C05431=1052.907,134.284,-84.781,171.313,33.859,156.345
C05432=1052.901,134.035,-84.760,171.311,33.857,156.345
C05433=1052.896,133.786,-84.739,171.310,33.854,156.344
C05434=1052.889,133.537,-84.718,171.307,33.852,156.344
C05435=1052.884,133.288,-84.697,171.305,33.850,156.344
C05436=1052.878,133.038,-84.676,171.303,33.847,156.343
C05437=1052.871,132.790,-84.656,171.301,33.845,156.343
C05438=1052.866,132.540,-84.635,171.300,33.843,156.342
C05439=1052.860,132.292,-84.613,171.298,33.841,156.342
C05440=1052.853,132.042,-84.593,171.296,33.838,156.342
C05441=1052.848,131.794,-84.572,171.294,33.836,156.341
C05442=1052.842,131.544,-84.551,171.293,33.834,156.341
C05443=1052.836,131.296,-84.530,171.291,33.832,156.340
C05444=1052.829,131.046,-84.510,171.289,33.829,156.340
C05445=1052.824,130.797,-84.489,171.287,33.827,156.340
C05446=1052.817,130.548,-84.468,171.286,33.825,156.339
C05447=1052.812,130.299,-84.448,171.284,33.823,156.339
C05448=1052.805,130.049,-84.427,171.282,33.821,156.339
C05449=1052.799,129.801,-84.407,171.280,33.818,156.338
C05450=1052.793,129.551,-84.386,171.279,33.816,156.338
C05451=1052.786,129.303,-84.365,171.277,33.814,156.337
C05452=1052.780,129.054,-84.345,171.275,33.812,156.337
C05453=1052.774,128.804,-84.324,171.273,33.809,156.337
C05454=1052.768,128.556,-84.303,171.271,33.807,156.336
C05455=1052.761,128.306,-84.283,171.269,33.806,156.336
C05456=1052.756,128.057,-84.262,171.267,33.803,156.336
C05457=1052.750,127.808,-84.242,171.265,33.801,156.335
C05458=1052.744,127.559,-84.221,171.263,33.798,156.335
C05459=1052.738,127.310,-84.201,171.262,33.797,156.334
C05460=1052.731,127.061,-84.180,171.260,33.794,156.334
C05461=1052.726,126.812,-84.159,171.258,33.792,156.334
C05462=1052.719,126.563,-84.139,171.257,33.790,156.333
C05463=1052.712,126.277,-84.115,171.255,33.788,156.333
C05464=1052.705,125.991,-84.092,171.253,33.785,156.332
C05465=1052.698,125.706,-84.069,171.251,33.782,156.332
C05466=1052.692,125.421,-84.045,171.249,33.780,156.332
C05467=1052.685,125.172,-84.025,171.247,33.777,156.331
C05468=1052.679,124.924,-84.004,171.245,33.775,156.331
C05469=1052.673,124.674,-83.983,171.243,33.773,156.330
C05470=1052.667,124.425,-83.963,171.242,33.771,156.330
C05471=1052.661,124.175,-83.943,171.240,33.768,156.330
C05472=1052.655,123.926,-83.923,171.238,33.766,156.329
C05473=1052.649,123.677,-83.903,171.236,33.764,156.329
C05474=1052.643,123.429,-83.882,171.235,33.762,156.328
C05475=1052.637,123.179,-83.861,171.232,33.760,156.328
C05476=1052.631,122.930,-83.841,171.230,33.757,156.328
C05477=1052.625,122.681,-83.821,171.229,33.755,156.327
C05478=1052.619,122.432,-83.801,171.227,33.753,156.327
C05479=1052.613,122.182,-83.780,171.225,33.751,156.327
C05480=1052.607,121.934,-83.760,171.223,33.748,156.326
C05481=1052.601,121.685,-83.740,171.222,33.746,156.326
C05482=1052.595,121.436,-83.718,171.220,33.744,156.325
C05483=1052.589,121.187,-83.698,171.218,33.742,156.325
C05484=1052.583,120.938,-83.678,171.217,33.739,156.325
C05485=1052.577,120.688,-83.657,171.215,33.737,156.324
C05486=1052.571,120.439,-83.637,171.213,33.735,156.324
C05487=1052.565,120.191,-83.617,171.211,33.733,156.324
C05488=1052.558,119.941,-83.597,171.210,33.731,156.323
C05489=1052.553,119.692,-83.577,171.208,33.728,156.323
C05490=1052.547,119.443,-83.557,171.206,33.726,156.322
C05491=1052.540,119.194,-83.536,171.205,33.724,156.322
C05492=1052.535,118.944,-83.516,171.203,33.722,156.322
C05493=1052.529,118.696,-83.496,171.201,33.719,156.321
C05494=1052.523,118.447,-83.476,171.200,33.718,156.321
C05495=1052.517,118.197,-83.456,171.198,33.715,156.321
C05496=1052.511,117.948,-83.435,171.196,33.713,156.320
C05497=1052.505,117.699,-83.415,171.194,33.710,156.320
C05498=1052.499,117.450,-83.395,171.192,33.708,156.319
C05499=1052.493,117.201,-83.374,171.190,33.706,156.319
C05500=1052.487,116.952,-83.354,171.188,33.704,156.319
C05501=1052.481,116.703,-83.334,171.187,33.701,156.318
C05502=1052.475,116.454,-83.314,171.185,33.699,156.318
C05503=1052.470,116.204,-83.294,171.183,33.697,156.317
C05504=1052.464,115.955,-83.274,171.182,33.695,156.317
C05505=1052.458,115.706,-83.254,171.180,33.692,156.317
C05506=1052.451,115.457,-83.234,171.178,33.690,156.316
C05507=1052.446,115.208,-83.213,171.177,33.688,156.316
C05508=1052.440,114.959,-83.193,171.175,33.686,156.316
C05509=1052.434,114.710,-83.173,171.173,33.683,156.315
C05510=1052.428,114.461,-83.153,171.172,33.682,156.315
C05511=1052.423,114.211,-83.133,171.170,33.679,156.314
C05512=1052.417,113.962,-83.113,171.168,33.677,156.314
C05513=1052.411,113.713,-83.093,171.167,33.674,156.314
C05514=1052.405,113.464,-83.073,171.165,33.672,156.313
C05515=1052.398,113.215,-83.053,171.163,33.670,156.313
C05516=1052.392,112.965,-83.034,171.161,33.668,156.313
C05517=1052.386,112.717,-83.014,171.160,33.666,156.312
C05518=1052.380,112.468,-82.994,171.158,33.663,156.312
C05519=1052.374,112.218,-82.973,171.156,33.661,156.311
C05520=1052.368,111.969,-82.954,171.155,33.659,156.311
C05521=1052.362,111.720,-82.934,171.153,33.657,156.311
C05522=1052.356,111.471,-82.914,171.151,33.655,156.310
C05523=1052.350,111.222,-82.894,171.149,33.653,156.310
C05524=1052.344,110.972,-82.875,171.147,33.651,156.310
C05525=1052.338,110.723,-82.855,171.145,33.648,156.309
C05526=1052.332,110.475,-82.835,171.144,33.646,156.309
C05527=1052.324,110.189,-82.813,171.142,33.643,156.308
C05528=1052.318,109.903,-82.790,171.140,33.641,156.308
C05529=1052.311,109.618,-82.768,171.138,33.639,156.308
C05530=1052.303,109.332,-82.745,171.136,33.636,156.307
C05531=1052.297,109.083,-82.725,171.134,33.634,156.307
C05532=1052.292,108.834,-82.706,171.133,33.632,156.306
C05533=1052.285,108.584,-82.686,171.131,33.630,156.306
C05534=1052.279,108.336,-82.666,171.129,33.627,156.306
C05535=1052.273,108.086,-82.647,171.128,33.625,156.305
C05536=1052.267,107.838,-82.627,171.126,33.623,156.305
C05537=1052.261,107.588,-82.608,171.124,33.621,156.305
C05538=1052.254,107.339,-82.588,171.123,33.619,156.304
C05539=1052.248,107.090,-82.568,171.121,33.617,156.304
C05540=1052.243,106.840,-82.548,171.119,33.614,156.304
C05541=1052.237,106.592,-82.528,171.117,33.612,156.303
C05542=1052.230,106.343,-82.510,171.116,33.610,156.303
C05543=1052.224,106.094,-82.490,171.114,33.608,156.302
C05544=1052.218,105.844,-82.470,171.112,33.606,156.302
C05545=1052.212,105.595,-82.450,171.111,33.603,156.302
C05546=1052.206,105.345,-82.431,171.109,33.601,156.301
C05547=1052.200,105.096,-82.411,171.108,33.600,156.301
C05548=1052.194,104.847,-82.392,171.106,33.597,156.301
C05549=1052.188,104.599,-82.372,171.104,33.595,156.300
C05550=1052.182,104.349,-82.353,171.103,33.593,156.300
C05551=1052.176,104.100,-82.333,171.101,33.590,156.299
C05552=1052.170,103.850,-82.314,171.098,33.589,156.299
C05553=1052.163,103.602,-82.294,171.097,33.586,156.299
C05554=1052.158,103.352,-82.275,171.095,33.584,156.298
C05555=1052.152,103.103,-82.255,171.093,33.582,156.298
C05556=1052.146,102.854,-82.236,171.092,33.580,156.298
C05557=1052.140,102.605,-82.217,171.090,33.578,156.297
C05558=1052.133,102.356,-82.197,171.088,33.576,156.297
C05559=1052.128,102.107,-82.178,171.087,33.573,156.297
C05560=1052.122,101.858,-82.158,171.085,33.571,156.296
C05561=1052.116,101.608,-82.139,171.083,33.568,156.296
C05562=1052.110,101.359,-82.120,171.082,33.567,156.295
C05563=1052.104,101.110,-82.100,171.080,33.565,156.295
C05564=1052.098,100.861,-82.081,171.078,33.562,156.295
C05565=1052.092,100.611,-82.061,171.077,33.560,156.294
C05566=1052.086,100.362,-82.041,171.075,33.558,156.294
C05567=1052.079,100.113,-82.023,171.073,33.556,156.294
C05568=1052.074,99.864,-82.003,171.072,33.554,156.293
C05569=1052.067,99.615,-81.984,171.070,33.552,156.293
C05570=1052.061,99.366,-81.965,171.068,33.549,156.293
C05571=1052.055,99.116,-81.946,171.067,33.547,156.292
C05572=1052.049,98.867,-81.927,171.065,33.545,156.292
C05573=1052.042,98.619,-81.908,171.063,33.543,156.292
C05574=1052.037,98.369,-81.888,171.062,33.541,156.291
C05575=1052.031,98.120,-81.869,171.060,33.539,156.291
C05576=1052.024,97.871,-81.850,171.059,33.537,156.291
C05577=1052.018,97.621,-81.830,171.057,33.534,156.290
C05578=1052.011,97.372,-81.811,171.055,33.532,156.290
C05579=1052.006,97.122,-81.792,171.054,33.530,156.289
C05580=1051.999,96.873,-81.774,171.052,33.528,156.289
C05581=1051.994,96.624,-81.754,171.050,33.526,156.289
C05582=1051.987,96.375,-81.735,171.049,33.524,156.288
C05583=1051.981,96.126,-81.716,171.047,33.522,156.288
C05584=1051.975,95.877,-81.697,171.045,33.519,156.288
C05585=1051.969,95.627,-81.678,171.044,33.517,156.287
C05586=1051.963,95.378,-81.659,171.042,33.515,156.287
C05587=1051.957,95.129,-81.639,171.040,33.513,156.287
C05588=1051.951,94.880,-81.620,171.038,33.511,156.286
C05589=1051.945,94.631,-81.601,171.036,33.509,156.286
C05590=1051.939,94.382,-81.582,171.034,33.506,156.285
C05591=1051.932,94.096,-81.561,171.033,33.504,156.285
C05592=1051.925,93.810,-81.538,171.031,33.502,156.285
C05593=1051.918,93.525,-81.517,171.029,33.499,156.284
C05594=1051.912,93.240,-81.495,171.027,33.497,156.284
C05595=1051.905,92.990,-81.477,171.025,33.495,156.283
C05596=1051.899,92.741,-81.457,171.024,33.493,156.283
C05597=1051.893,92.492,-81.439,171.022,33.490,156.283
C05598=1051.887,92.242,-81.419,171.020,33.488,156.282
C05599=1051.881,91.994,-81.400,171.019,33.486,156.282
C05600=1051.875,91.745,-81.381,171.017,33.484,156.282
C05601=1051.868,91.495,-81.362,171.016,33.482,156.281
C05602=1051.863,91.246,-81.343,171.014,33.480,156.281
C05603=1051.856,90.997,-81.324,171.012,33.477,156.281
C05604=1051.851,90.747,-81.305,171.011,33.475,156.280
C05605=1051.844,90.498,-81.286,171.009,33.473,156.280
C05606=1051.838,90.249,-81.268,171.007,33.471,156.280
C05607=1051.832,90.000,-81.249,171.006,33.469,156.279
C05608=1051.826,89.750,-81.231,171.004,33.467,156.279
C05609=1051.820,89.501,-81.212,171.002,33.465,156.279
C05610=1051.813,89.252,-81.193,171.001,33.463,156.278
C05611=1051.807,89.002,-81.174,170.999,33.460,156.278
C05612=1051.802,88.754,-81.156,170.998,33.458,156.277
C05613=1051.795,88.505,-81.137,170.996,33.456,156.277
C05614=1051.789,88.256,-81.118,170.994,33.454,156.277
C05615=1051.783,88.006,-81.099,170.993,33.452,156.276
C05616=1051.777,87.757,-81.081,170.991,33.450,156.276
C05617=1051.770,87.508,-81.062,170.989,33.448,156.276
C05618=1051.764,87.259,-81.043,170.988,33.446,156.275
C05619=1051.758,87.009,-81.025,170.986,33.444,156.275
C05620=1051.752,86.760,-81.006,170.984,33.441,156.275
C05621=1051.746,86.511,-80.987,170.983,33.439,156.274
C05622=1051.739,86.261,-80.969,170.981,33.437,156.274
C05623=1051.733,86.012,-80.950,170.979,33.435,156.274
C05624=1051.727,85.763,-80.931,170.978,33.433,156.273
C05625=1051.722,85.514,-80.913,170.976,33.431,156.273
C05626=1051.715,85.265,-80.895,170.975,33.429,156.273
C05627=1051.709,85.016,-80.876,170.973,33.427,156.272
C05628=1051.703,84.766,-80.857,170.971,33.424,156.272
C05629=1051.697,84.517,-80.838,170.970,33.422,156.272
C05630=1051.690,84.267,-80.820,170.968,33.420,156.271
C05631=1051.684,84.018,-80.802,170.966,33.418,156.271
C05632=1051.678,83.769,-80.782,170.965,33.416,156.270
C05633=1051.672,83.520,-80.764,170.963,33.414,156.270
C05634=1051.666,83.271,-80.746,170.962,33.412,156.270
C05635=1051.660,83.021,-80.727,170.960,33.410,156.270
C05636=1051.654,82.772,-80.709,170.958,33.407,156.269
C05637=1051.648,82.523,-80.690,170.957,33.405,156.269
C05638=1051.642,82.273,-80.672,170.954,33.403,156.268
C05639=1051.636,82.025,-80.653,170.952,33.401,156.268
C05640=1051.629,81.776,-80.635,170.951,33.399,156.268
C05641=1051.623,81.526,-80.617,170.949,33.397,156.267
C05642=1051.618,81.276,-80.598,170.948,33.395,156.267
C05643=1051.611,81.027,-80.579,170.946,33.392,156.267
C05644=1051.606,80.778,-80.561,170.944,33.390,156.266
C05645=1051.599,80.529,-80.543,170.943,33.389,156.266
C05646=1051.593,80.280,-80.524,170.941,33.387,156.266
C05647=1051.587,80.030,-80.506,170.939,33.384,156.265
C05648=1051.581,79.781,-80.487,170.938,33.382,156.265
C05649=1051.575,79.532,-80.469,170.936,33.380,156.265
C05650=1051.569,79.283,-80.451,170.935,33.378,156.264
C05651=1051.563,79.034,-80.432,170.933,33.375,156.264
C05652=1051.557,78.784,-80.414,170.931,33.373,156.264
C05653=1051.551,78.535,-80.396,170.930,33.372,156.263
C05654=1051.545,78.286,-80.377,170.928,33.369,156.263
C05655=1051.538,78.001,-80.356,170.926,33.367,156.262
C05656=1051.530,77.715,-80.335,170.924,33.364,156.262
C05657=1051.524,77.428,-80.314,170.923,33.362,156.262
C05658=1051.516,77.143,-80.294,170.921,33.360,156.261
C05659=1051.510,76.894,-80.275,170.919,33.358,156.261
C05660=1051.504,76.645,-80.257,170.917,33.355,156.261
C05661=1051.498,76.396,-80.239,170.916,33.353,156.260
C05662=1051.492,76.146,-80.221,170.914,33.351,156.260
C05663=1051.485,75.897,-80.202,170.913,33.349,156.260
C05664=1051.479,75.647,-80.184,170.911,33.347,156.259
C05665=1051.474,75.399,-80.166,170.909,33.345,156.259
C05666=1051.467,75.149,-80.148,170.908,33.343,156.259
C05667=1051.461,74.900,-80.129,170.906,33.341,156.258
C05668=1051.455,74.650,-80.111,170.904,33.339,156.258
C05669=1051.449,74.402,-80.093,170.903,33.337,156.258
C05670=1051.443,74.152,-80.075,170.901,33.335,156.257
C05671=1051.436,73.903,-80.058,170.900,33.332,156.257
C05672=1051.430,73.654,-80.039,170.898,33.330,156.257
C05673=1051.424,73.404,-80.022,170.896,33.328,156.256
C05674=1051.418,73.155,-80.003,170.895,33.326,156.256
C05675=1051.412,72.906,-79.985,170.893,33.324,156.256
C05676=1051.406,72.657,-79.967,170.891,33.322,156.255
C05677=1051.400,72.407,-79.949,170.890,33.320,156.255
C05678=1051.394,72.158,-79.931,170.888,33.318,156.254
C05679=1051.387,71.909,-79.912,170.887,33.316,156.254
C05680=1051.382,71.660,-79.895,170.885,33.314,156.254
C05681=1051.375,71.410,-79.877,170.883,33.311,156.253
C05682=1051.368,71.161,-79.859,170.882,33.309,156.253
C05683=1051.363,70.912,-79.841,170.880,33.307,156.253
C05684=1051.357,70.662,-79.823,170.878,33.305,156.252
C05685=1051.350,70.413,-79.805,170.877,33.304,156.252
C05686=1051.345,70.164,-79.787,170.875,33.301,156.252
C05687=1051.339,69.914,-79.769,170.874,33.299,156.251
C05688=1051.332,69.665,-79.750,170.872,33.297,156.251
C05689=1051.326,69.416,-79.733,170.870,33.295,156.251
C05690=1051.320,69.167,-79.716,170.869,33.293,156.250
C05691=1051.314,68.917,-79.698,170.867,33.291,156.250
C05692=1051.308,68.669,-79.679,170.865,33.288,156.250
C05693=1051.301,68.419,-79.662,170.864,33.287,156.249
C05694=1051.295,68.169,-79.644,170.862,33.285,156.249
C05695=1051.289,67.920,-79.626,170.861,33.283,156.249
C05696=1051.283,67.671,-79.609,170.859,33.281,156.248
C05697=1051.276,67.422,-79.591,170.857,33.279,156.248
C05698=1051.271,67.173,-79.573,170.856,33.277,156.248
C05699=1051.264,66.923,-79.555,170.854,33.274,156.247
C05700=1051.258,66.673,-79.537,170.852,33.272,156.247
C05701=1051.252,66.425,-79.520,170.851,33.270,156.247
C05702=1051.246,66.175,-79.501,170.849,33.268,156.246
C05703=1051.240,65.926,-79.484,170.847,33.266,156.246
C05704=1051.233,65.677,-79.467,170.846,33.264,156.246
C05705=1051.227,65.427,-79.449,170.844,33.262,156.245
C05706=1051.222,65.178,-79.431,170.843,33.260,156.245
C05707=1051.215,64.929,-79.414,170.841,33.258,156.245
C05708=1051.209,64.679,-79.396,170.839,33.256,156.244
C05709=1051.203,64.430,-79.378,170.838,33.254,156.244
C05710=1051.197,64.181,-79.360,170.836,33.252,156.244
C05711=1051.190,63.932,-79.343,170.834,33.250,156.243
C05712=1051.184,63.683,-79.325,170.833,33.248,156.243
C05713=1051.177,63.433,-79.307,170.831,33.246,156.243
C05714=1051.171,63.184,-79.290,170.830,33.244,156.243
C05715=1051.165,62.934,-79.272,170.828,33.242,156.242
C05716=1051.158,62.685,-79.255,170.826,33.240,156.242
C05717=1051.153,62.436,-79.238,170.825,33.238,156.242
C05718=1051.146,62.187,-79.220,170.823,33.236,156.241
C05719=1051.139,61.901,-79.200,170.821,33.233,156.241
C05720=1051.132,61.615,-79.180,170.819,33.231,156.241
C05721=1051.124,61.330,-79.160,170.817,33.229,156.240
C05722=1051.117,61.044,-79.140,170.815,33.227,156.240
C05723=1051.111,60.794,-79.122,170.814,33.225,156.239
C05724=1051.105,60.545,-79.105,170.812,33.223,156.239
C05725=1051.098,60.296,-79.087,170.810,33.221,156.239
C05726=1051.092,60.046,-79.070,170.809,33.219,156.239
C05727=1051.085,59.797,-79.053,170.807,33.217,156.238
C05728=1051.080,59.547,-79.036,170.806,33.215,156.238
C05729=1051.073,59.298,-79.019,170.804,33.213,156.238
C05730=1051.067,59.049,-79.001,170.802,33.211,156.237
C05731=1051.061,58.800,-78.984,170.801,33.208,156.237
C05732=1051.054,58.550,-78.967,170.799,33.206,156.237
C05733=1051.048,58.301,-78.949,170.797,33.204,156.236
C05734=1051.042,58.052,-78.932,170.796,33.202,156.236
C05735=1051.036,57.802,-78.914,170.794,33.200,156.236
C05736=1051.029,57.553,-78.897,170.792,33.198,156.235
C05737=1051.023,57.303,-78.880,170.791,33.196,156.235
C05738=1051.017,57.054,-78.863,170.789,33.194,156.235
C05739=1051.010,56.805,-78.845,170.787,33.192,156.234
C05740=1051.005,56.556,-78.828,170.786,33.190,156.234
C05741=1050.998,56.306,-78.810,170.784,33.188,156.234
C05742=1050.992,56.058,-78.793,170.783,33.186,156.233
C05743=1050.986,55.807,-78.776,170.781,33.184,156.233
C05744=1050.980,55.559,-78.759,170.779,33.182,156.233
C05745=1050.974,55.309,-78.741,170.778,33.180,156.232
C05746=1050.967,55.060,-78.724,170.776,33.178,156.232
C05747=1050.960,54.811,-78.707,170.774,33.176,156.232
C05748=1050.955,54.561,-78.690,170.773,33.174,156.231
C05749=1050.948,54.312,-78.673,170.771,33.172,156.231
C05750=1050.943,54.063,-78.655,170.769,33.170,156.231
C05751=1050.936,53.813,-78.638,170.768,33.168,156.230
C05752=1050.930,53.564,-78.622,170.766,33.166,156.230
C05753=1050.924,53.314,-78.604,170.765,33.164,156.230
C05754=1050.918,53.065,-78.587,170.763,33.162,156.229
C05755=1050.911,52.816,-78.569,170.761,33.160,156.229
C05756=1050.906,52.566,-78.553,170.760,33.158,156.229
C05757=1050.899,52.317,-78.535,170.758,33.156,156.229
C05758=1050.892,52.068,-78.518,170.756,33.154,156.228
C05759=1050.887,51.818,-78.501,170.755,33.152,156.228
C05760=1050.880,51.569,-78.484,170.753,33.150,156.228
C05761=1050.875,51.320,-78.467,170.751,33.148,156.227
C05762=1050.868,51.070,-78.450,170.750,33.146,156.227
C05763=1050.862,50.821,-78.433,170.748,33.144,156.227
C05764=1050.856,50.571,-78.415,170.747,33.141,156.226
C05765=1050.850,50.322,-78.399,170.745,33.139,156.226
C05766=1050.844,50.073,-78.382,170.743,33.137,156.226
C05767=1050.838,49.824,-78.364,170.742,33.136,156.225
C05768=1050.832,49.574,-78.348,170.740,33.133,156.225
C05769=1050.825,49.325,-78.330,170.738,33.131,156.225
C05770=1050.819,49.076,-78.313,170.737,33.130,156.224
C05771=1050.813,48.827,-78.296,170.735,33.128,156.224
C05772=1050.806,48.577,-78.279,170.733,33.125,156.224
C05773=1050.801,48.327,-78.262,170.732,33.124,156.223
C05774=1050.795,48.079,-78.245,170.730,33.122,156.223
C05775=1050.788,47.829,-78.228,170.728,33.119,156.223
C05776=1050.783,47.580,-78.211,170.727,33.117,156.222
C05777=1050.777,47.331,-78.194,170.725,33.115,156.222
C05778=1050.770,47.081,-78.177,170.724,33.113,156.222
C05779=1050.765,46.832,-78.160,170.722,33.111,156.221
C05780=1050.759,46.582,-78.144,170.720,33.109,156.221
C05781=1050.752,46.333,-78.126,170.719,33.107,156.221
C05782=1050.747,46.083,-78.109,170.717,33.105,156.220
C05783=1050.739,45.798,-78.090,170.715,33.102,156.220
C05784=1050.732,45.511,-78.071,170.713,33.100,156.220
C05785=1050.725,45.225,-78.051,170.711,33.098,156.219
C05786=1050.718,44.939,-78.032,170.710,33.095,156.219
C05787=1050.712,44.690,-78.015,170.708,33.093,156.219
C05788=1050.706,44.441,-77.998,170.706,33.091,156.218
C05789=1050.700,44.191,-77.981,170.705,33.089,156.218
C05790=1050.694,43.942,-77.964,170.703,33.087,156.218
C05791=1050.688,43.693,-77.947,170.701,33.085,156.217
C05792=1050.682,43.443,-77.931,170.700,33.083,156.217
C05793=1050.675,43.194,-77.914,170.698,33.081,156.217
C05794=1050.669,42.945,-77.897,170.696,33.079,156.216
C05795=1050.663,42.695,-77.881,170.695,33.077,156.216
C05796=1050.656,42.446,-77.864,170.693,33.075,156.216
C05797=1050.651,42.197,-77.848,170.691,33.073,156.215
C05798=1050.645,41.947,-77.831,170.690,33.071,156.215
C05799=1050.638,41.697,-77.813,170.688,33.069,156.215
C05800=1050.632,41.448,-77.797,170.686,33.067,156.215
C05801=1050.627,41.199,-77.781,170.685,33.065,156.214
C05802=1050.620,40.949,-77.764,170.683,33.063,156.214
C05803=1050.614,40.700,-77.747,170.681,33.061,156.214
C05804=1050.608,40.451,-77.731,170.680,33.059,156.213
C05805=1050.602,40.202,-77.714,170.678,33.057,156.213
C05806=1050.595,39.952,-77.697,170.676,33.055,156.213
C05807=1050.589,39.702,-77.681,170.675,33.053,156.212
C05808=1050.583,39.454,-77.664,170.673,33.051,156.212
C05809=1050.576,39.204,-77.648,170.671,33.049,156.212
C05810=1050.570,38.954,-77.631,170.670,33.047,156.211
C05811=1050.564,38.705,-77.615,170.668,33.045,156.211
C05812=1050.558,38.456,-77.598,170.667,33.043,156.211
C05813=1050.551,38.206,-77.581,170.665,33.041,156.211
C05814=1050.546,37.957,-77.565,170.663,33.039,156.210
C05815=1050.540,37.708,-77.549,170.662,33.037,156.210
C05816=1050.533,37.459,-77.532,170.660,33.035,156.210
C05817=1050.527,37.209,-77.515,170.658,33.033,156.209
C05818=1050.521,36.959,-77.499,170.657,33.031,156.209
C05819=1050.515,36.710,-77.483,170.655,33.029,156.209
C05820=1050.509,36.461,-77.467,170.653,33.027,156.208
C05821=1050.502,36.211,-77.450,170.651,33.025,156.208
C05822=1050.495,35.962,-77.434,170.650,33.024,156.208
C05823=1050.489,35.713,-77.417,170.648,33.022,156.208
C05824=1050.483,35.464,-77.401,170.646,33.020,156.207
C05825=1050.477,35.213,-77.384,170.645,33.018,156.207
C05826=1050.471,34.964,-77.368,170.644,33.016,156.207
C05827=1050.465,34.715,-77.352,170.642,33.014,156.206
C05828=1050.458,34.466,-77.336,170.641,33.012,156.206
C05829=1050.452,34.216,-77.320,170.639,33.010,156.206
C05830=1050.446,33.967,-77.303,170.637,33.008,156.205
C05831=1050.440,33.718,-77.286,170.636,33.006,156.205
C05832=1050.434,33.468,-77.270,170.634,33.004,156.205
C05833=1050.428,33.219,-77.254,170.632,33.002,156.205
C05834=1050.420,32.969,-77.238,170.631,33.001,156.204
C05835=1050.414,32.720,-77.222,170.629,32.998,156.204
C05836=1050.408,32.471,-77.205,170.627,32.996,156.204
C05837=1050.403,32.221,-77.189,170.626,32.995,156.203
C05838=1050.397,31.972,-77.173,170.624,32.992,156.203
C05839=1050.390,31.723,-77.157,170.622,32.990,156.203
C05840=1050.383,31.473,-77.141,170.621,32.988,156.202
C05841=1050.377,31.223,-77.124,170.619,32.986,156.202
C05842=1050.371,30.974,-77.108,170.617,32.984,156.202
C05843=1050.365,30.725,-77.092,170.615,32.983,156.202
C05844=1050.359,30.476,-77.076,170.614,32.981,156.201
C05845=1050.353,30.226,-77.060,170.612,32.979,156.201
C05846=1050.346,29.976,-77.043,170.610,32.977,156.201
C05847=1050.340,29.691,-77.025,170.609,32.974,156.200
C05848=1050.332,29.404,-77.006,170.607,32.972,156.200
C05849=1050.325,29.119,-76.988,170.605,32.970,156.200
C05850=1050.318,28.833,-76.969,170.603,32.968,156.199
C05851=1050.312,28.583,-76.953,170.601,32.966,156.199
C05852=1050.306,28.333,-76.938,170.599,32.964,156.199
C05853=1050.299,28.084,-76.922,170.598,32.962,156.198
C05854=1050.293,27.834,-76.905,170.596,32.960,156.198
C05855=1050.287,27.585,-76.889,170.594,32.958,156.198
C05856=1050.280,27.336,-76.873,170.593,32.956,156.197
C05857=1050.274,27.087,-76.857,170.591,32.955,156.197
C05858=1050.269,26.837,-76.841,170.589,32.953,156.197
C05859=1050.262,26.588,-76.825,170.587,32.951,156.197
C05860=1050.256,26.338,-76.810,170.586,32.949,156.196
C05861=1050.250,26.088,-76.793,170.584,32.947,156.196
C05862=1050.243,25.839,-76.777,170.582,32.945,156.196
C05863=1050.237,25.590,-76.761,170.581,32.943,156.196
C05864=1050.230,25.341,-76.746,170.579,32.941,156.195
C05865=1050.225,25.091,-76.730,170.577,32.939,156.195
C05866=1050.218,24.842,-76.714,170.576,32.937,156.195
C05867=1050.212,24.592,-76.698,170.574,32.935,156.194
C05868=1050.206,24.343,-76.682,170.572,32.934,156.194
C05869=1050.199,24.094,-76.666,170.570,32.932,156.194
C05870=1050.194,23.844,-76.651,170.569,32.930,156.193
C05871=1050.186,23.594,-76.635,170.567,32.928,156.193
C05872=1050.181,23.345,-76.618,170.565,32.926,156.193
C05873=1050.174,23.096,-76.603,170.564,32.924,156.193
C05874=1050.168,22.846,-76.587,170.562,32.923,156.192
C05875=1050.162,22.597,-76.571,170.560,32.920,156.192
C05876=1050.156,22.348,-76.555,170.558,32.918,156.192
C05877=1050.150,22.098,-76.540,170.558,32.917,156.191
C05878=1050.143,21.849,-76.524,170.556,32.914,156.191
C05879=1050.137,21.599,-76.508,170.554,32.913,156.191
C05880=1050.131,21.350,-76.493,170.553,32.911,156.191
C05881=1050.125,21.100,-76.477,170.551,32.909,156.190
C05882=1050.118,20.851,-76.461,170.549,32.907,156.190
C05883=1050.113,20.601,-76.445,170.547,32.905,156.190
C05884=1050.106,20.352,-76.430,170.546,32.904,156.190
C05885=1050.100,20.103,-76.413,170.544,32.902,156.189
C05886=1050.094,19.853,-76.398,170.542,32.900,156.189
C05887=1050.088,19.604,-76.382,170.541,32.898,156.189
C05888=1050.081,19.355,-76.367,170.539,32.896,156.188
C05889=1050.075,19.105,-76.351,170.537,32.894,156.188
C05890=1050.069,18.856,-76.335,170.535,32.892,156.188
C05891=1050.063,18.606,-76.320,170.534,32.890,156.187
C05892=1050.056,18.357,-76.304,170.532,32.888,156.187
C05893=1050.050,18.107,-76.289,170.530,32.887,156.187
C05894=1050.044,17.858,-76.273,170.528,32.885,156.187
C05895=1050.037,17.609,-76.257,170.527,32.883,156.186
C05896=1050.032,17.359,-76.242,170.525,32.881,156.186
C05897=1050.025,17.110,-76.226,170.523,32.879,156.186
C05898=1050.019,16.860,-76.211,170.522,32.877,156.186
C05899=1050.013,16.611,-76.195,170.520,32.875,156.185
C05900=1050.006,16.361,-76.180,170.518,32.873,156.185
C05901=1050.000,16.112,-76.164,170.516,32.872,156.185
C05902=1049.994,15.862,-76.149,170.515,32.870,156.184
C05903=1049.987,15.613,-76.133,170.513,32.868,156.184
C05904=1049.982,15.363,-76.118,170.511,32.866,156.184
C05905=1049.975,15.114,-76.102,170.509,32.864,156.184
C05906=1049.968,14.864,-76.087,170.508,32.862,156.183
C05907=1049.962,14.615,-76.071,170.506,32.860,156.183
C05908=1049.956,14.365,-76.056,170.504,32.858,156.183
C05909=1049.950,14.115,-76.040,170.502,32.857,156.183
C05910=1049.944,13.866,-76.024,170.501,32.855,156.182
C05911=1049.937,13.582,-76.007,170.499,32.853,156.182
C05912=1049.929,13.297,-75.990,170.497,32.851,156.182
C05913=1049.922,13.012,-75.972,170.495,32.849,156.181
C05914=1049.915,12.728,-75.955,170.493,32.847,156.181
C05915=1049.909,12.478,-75.940,170.491,32.845,156.181
C05916=1049.902,12.229,-75.924,170.490,32.843,156.181
C05917=1049.896,11.979,-75.909,170.488,32.841,156.180
C05918=1049.890,11.730,-75.894,170.487,32.840,156.180
C05919=1049.883,11.481,-75.879,170.485,32.838,156.180
C05920=1049.877,11.231,-75.864,170.483,32.836,156.179
C05921=1049.871,10.981,-75.848,170.481,32.834,156.179
C05922=1049.864,10.732,-75.833,170.480,32.832,156.179
C05923=1049.858,10.482,-75.818,170.478,32.831,156.179
C05924=1049.851,10.233,-75.803,170.476,32.829,156.178
C05925=1049.845,9.983,-75.788,170.474,32.827,156.178
C05926=1049.838,9.734,-75.772,170.472,32.825,156.178
C05927=1049.832,9.484,-75.757,170.471,32.823,156.178
C05928=1049.827,9.235,-75.742,170.469,32.822,156.177
C05929=1049.820,8.986,-75.726,170.467,32.820,156.177
C05930=1049.814,8.736,-75.711,170.465,32.818,156.177
C05931=1049.807,8.487,-75.696,170.464,32.817,156.177
C05932=1049.801,8.237,-75.681,170.462,32.814,156.176
C05933=1049.795,7.987,-75.666,170.460,32.812,156.176
C05934=1049.788,7.738,-75.651,170.458,32.811,156.176
C05935=1049.782,7.489,-75.636,170.457,32.809,156.176
C05936=1049.777,7.239,-75.621,170.455,32.808,156.175
C05937=1049.770,6.990,-75.606,170.453,32.806,156.175
C05938=1049.764,6.740,-75.591,170.451,32.803,156.175
C05939=1049.757,6.491,-75.575,170.449,32.802,156.175
C05940=1049.751,6.241,-75.560,170.448,32.800,156.174
C05941=1049.744,5.992,-75.545,170.446,32.799,156.174
C05942=1049.739,5.743,-75.531,170.444,32.797,156.174
C05943=1049.732,5.493,-75.516,170.442,32.795,156.174
C05944=1049.726,5.243,-75.501,170.441,32.793,156.173
C05945=1049.719,4.994,-75.485,170.439,32.791,156.173
C05946=1049.713,4.744,-75.470,170.437,32.789,156.173
C05947=1049.707,4.495,-75.455,170.435,32.788,156.173
C05948=1049.701,4.246,-75.440,170.434,32.786,156.172
C05949=1049.695,3.996,-75.425,170.433,32.784,156.172
C05950=1049.689,3.746,-75.410,170.431,32.782,156.172
C05951=1049.682,3.497,-75.395,170.429,32.780,156.171
C05952=1049.676,3.248,-75.381,170.427,32.779,156.171
C05953=1049.670,2.998,-75.366,170.426,32.777,156.171
C05954=1049.664,2.749,-75.351,170.424,32.775,156.171
C05955=1049.657,2.499,-75.336,170.422,32.773,156.170
C05956=1049.651,2.250,-75.321,170.420,32.771,156.170
C05957=1049.645,2.001,-75.306,170.418,32.770,156.170
C05958=1049.638,1.751,-75.291,170.417,32.768,156.170
C05959=1049.633,1.501,-75.275,170.415,32.766,156.169
C05960=1049.627,1.252,-75.261,170.413,32.764,156.169
C05961=1049.621,1.003,-75.246,170.411,32.762,156.169
C05962=1049.614,0.753,-75.231,170.409,32.761,156.169
C05963=1049.608,0.503,-75.216,170.408,32.759,156.168
C05964=1049.602,0.254,-75.201,170.406,32.757,156.168
C05965=1049.596,0.005,-75.186,170.404,32.755,156.168
C05966=1049.589,-0.245,-75.171,170.402,32.753,156.168
C05967=1049.584,-0.495,-75.157,170.400,32.752,156.167
C05968=1049.577,-0.744,-75.142,170.399,32.750,156.167
C05969=1049.571,-0.994,-75.127,170.397,32.748,156.167
C05970=1049.565,-1.244,-75.112,170.395,32.746,156.167
C05971=1049.559,-1.492,-75.098,170.393,32.744,156.166
C05972=1049.552,-1.742,-75.083,170.392,32.743,156.166
C05973=1049.546,-1.992,-75.068,170.390,32.741,156.166
C05974=1049.540,-2.241,-75.053,170.388,32.739,156.166
C05975=1049.533,-2.524,-75.036,170.386,32.737,156.165
C05976=1049.527,-2.807,-75.020,170.384,32.735,156.165
C05977=1049.520,-3.090,-75.003,170.383,32.733,156.165
C05978=1049.513,-3.373,-74.986,170.381,32.731,156.164
C05979=1049.507,-3.622,-74.972,170.379,32.729,156.164
C05980=1049.500,-3.871,-74.957,170.377,32.728,156.164
C05981=1049.493,-4.121,-74.942,170.375,32.726,156.164
C05982=1049.487,-4.371,-74.928,170.373,32.724,156.163
C05983=1049.482,-4.620,-74.914,170.372,32.723,156.163
C05984=1049.474,-4.870,-74.899,170.370,32.721,156.163
C05985=1049.468,-5.119,-74.884,170.368,32.719,156.163
C05986=1049.462,-5.368,-74.870,170.366,32.717,156.162
C05987=1049.456,-5.618,-74.855,170.364,32.716,156.162
C05988=1049.449,-5.868,-74.841,170.362,32.714,156.162
C05989=1049.443,-6.117,-74.827,170.361,32.713,156.162
C05990=1049.437,-6.366,-74.812,170.359,32.711,156.162
C05991=1049.430,-6.616,-74.798,170.357,32.709,156.161
C05992=1049.424,-6.865,-74.783,170.355,32.708,156.161
C05993=1049.418,-7.115,-74.769,170.353,32.706,156.161
C05994=1049.412,-7.365,-74.754,170.351,32.704,156.161
C05995=1049.405,-7.614,-74.740,170.350,32.703,156.160
C05996=1049.399,-7.864,-74.725,170.348,32.701,156.160
C05997=1049.393,-8.113,-74.710,170.346,32.699,156.160
C05998=1049.386,-8.362,-74.697,170.344,32.697,156.160
C05999=1049.380,-8.612,-74.682,170.342,32.696,156.160
C06000=1049.374,-8.861,-74.668,170.340,32.694,156.159
C06001=1049.368,-9.111,-74.653,170.338,32.692,156.159
C06002=1049.361,-9.361,-74.639,170.337,32.691,156.159
C06003=1049.355,-9.610,-74.624,170.336,32.689,156.159
C06004=1049.349,-9.860,-74.610,170.334,32.687,156.158
C06005=1049.342,-10.109,-74.596,170.332,32.686,156.158
C06006=1049.336,-10.358,-74.581,170.330,32.684,156.158
C06007=1049.330,-10.608,-74.567,170.328,32.682,156.158
C06008=1049.324,-10.857,-74.553,170.327,32.680,156.157
C06009=1049.318,-11.107,-74.539,170.325,32.679,156.157
C06010=1049.312,-11.356,-74.524,170.323,32.678,156.157
C06011=1049.306,-11.607,-74.510,170.321,32.675,156.157
C06012=1049.299,-11.856,-74.496,170.319,32.674,156.157
C06013=1049.293,-12.105,-74.481,170.317,32.672,156.156
C06014=1049.287,-12.355,-74.467,170.315,32.671,156.156
C06015=1049.280,-12.604,-74.453,170.314,32.669,156.156
C06016=1049.274,-12.854,-74.439,170.312,32.667,156.156
C06017=1049.268,-13.103,-74.424,170.310,32.666,156.155
C06018=1049.262,-13.353,-74.410,170.308,32.664,156.155
C06019=1049.256,-13.602,-74.396,170.306,32.662,156.155
C06020=1049.250,-13.852,-74.382,170.304,32.661,156.155
C06021=1049.243,-14.101,-74.368,170.302,32.659,156.154
C06022=1049.237,-14.351,-74.353,170.301,32.657,156.154
C06023=1049.231,-14.600,-74.339,170.299,32.656,156.154
C06024=1049.224,-14.850,-74.325,170.297,32.654,156.154
C06025=1049.219,-15.099,-74.311,170.295,32.652,156.154
C06026=1049.212,-15.349,-74.297,170.293,32.650,156.153
C06027=1049.206,-15.599,-74.283,170.292,32.649,156.153
C06028=1049.199,-15.848,-74.269,170.290,32.647,156.153
C06029=1049.193,-16.098,-74.255,170.288,32.646,156.153
C06030=1049.187,-16.347,-74.241,170.286,32.644,156.152
C06031=1049.181,-16.597,-74.226,170.285,32.643,156.152
C06032=1049.174,-16.846,-74.213,170.283,32.641,156.152
C06033=1049.168,-17.096,-74.198,170.281,32.640,156.152
C06034=1049.162,-17.345,-74.185,170.279,32.638,156.152
C06035=1049.155,-17.595,-74.171,170.277,32.636,156.151
C06036=1049.149,-17.844,-74.157,170.275,32.635,156.151
C06037=1049.142,-18.094,-74.143,170.273,32.633,156.151
C06038=1049.137,-18.343,-74.128,170.271,32.632,156.151
C06039=1049.130,-18.584,-74.116,170.270,32.630,156.151
C06040=1049.125,-18.825,-74.102,170.268,32.628,156.150
C06041=1049.118,-19.066,-74.089,170.266,32.627,156.150
C06042=1049.112,-19.307,-74.075,170.264,32.625,156.150
C06043=1049.106,-19.548,-74.062,170.262,32.624,156.150
C06044=1049.100,-19.788,-74.048,170.260,32.623,156.150
C06045=1049.094,-20.029,-74.035,170.259,32.621,156.149
C06046=1049.088,-20.270,-74.022,170.257,32.619,156.149
C06047=1049.081,-20.519,-74.008,170.255,32.618,156.149
C06048=1049.075,-20.769,-73.994,170.253,32.616,156.149
C06049=1049.069,-21.019,-73.980,170.251,32.615,156.149
C06050=1049.064,-21.268,-73.966,170.249,32.613,156.148
C06051=1049.056,-21.518,-73.952,170.248,32.611,156.148
C06052=1049.050,-21.767,-73.939,170.246,32.610,156.148
C06053=1049.044,-22.017,-73.925,170.244,32.608,156.148
C06054=1049.038,-22.266,-73.911,170.242,32.607,156.148
C06055=1049.032,-22.516,-73.896,170.241,32.606,156.147
C06056=1049.025,-22.765,-73.883,170.239,32.603,156.147
C06057=1049.019,-23.015,-73.870,170.237,32.602,156.147
C06058=1049.013,-23.265,-73.856,170.235,32.601,156.147
C06059=1049.007,-23.514,-73.842,170.233,32.599,156.147
C06060=1049.001,-23.764,-73.828,170.231,32.598,156.146
C06061=1048.994,-24.013,-73.814,170.229,32.596,156.146
C06062=1048.988,-24.262,-73.801,170.227,32.594,156.146
C06063=1048.982,-24.513,-73.787,170.225,32.593,156.146
C06064=1048.976,-24.762,-73.773,170.223,32.591,156.146
C06065=1048.970,-25.011,-73.760,170.221,32.590,156.145
C06066=1048.963,-25.261,-73.746,170.219,32.588,156.145
C06067=1048.957,-25.511,-73.733,170.218,32.586,156.145
C06068=1048.951,-25.760,-73.719,170.216,32.585,156.145
C06069=1048.945,-26.010,-73.704,170.214,32.583,156.144
C06070=1048.938,-26.259,-73.691,170.212,32.582,156.144
C06071=1048.933,-26.508,-73.677,170.210,32.580,156.144
C06072=1048.926,-26.758,-73.664,170.208,32.578,156.144
C06073=1048.920,-27.008,-73.650,170.207,32.577,156.144
C06074=1048.914,-27.257,-73.637,170.205,32.576,156.143
C06075=1048.907,-27.507,-73.623,170.203,32.574,156.143
C06076=1048.901,-27.756,-73.609,170.201,32.573,156.143
C06077=1048.895,-28.006,-73.596,170.199,32.571,156.143
C06078=1048.888,-28.256,-73.583,170.197,32.570,156.143
C06079=1048.882,-28.505,-73.569,170.195,32.568,156.143
C06080=1048.876,-28.754,-73.556,170.193,32.567,156.142
C06081=1048.869,-29.004,-73.542,170.191,32.565,156.142
C06082=1048.863,-29.253,-73.529,170.189,32.564,156.142
C06083=1048.857,-29.503,-73.515,170.187,32.562,156.142
C06084=1048.851,-29.753,-73.502,170.186,32.561,156.142
C06085=1048.845,-30.003,-73.489,170.184,32.560,156.141
C06086=1048.839,-30.252,-73.476,170.182,32.558,156.141
C06087=1048.832,-30.502,-73.462,170.180,32.557,156.141
C06088=1048.826,-30.751,-73.449,170.178,32.555,156.141
C06089=1048.819,-31.001,-73.436,170.176,32.554,156.141
C06090=1048.812,-31.251,-73.422,170.174,32.552,156.141
C06091=1048.806,-31.500,-73.409,170.172,32.551,156.140
C06092=1048.801,-31.749,-73.395,170.170,32.549,156.140
C06093=1048.795,-31.999,-73.382,170.168,32.548,156.140
C06094=1048.788,-32.249,-73.368,170.167,32.546,156.140
C06095=1048.782,-32.498,-73.355,170.165,32.545,156.140
C06096=1048.776,-32.748,-73.342,170.163,32.544,156.139
C06097=1048.769,-32.997,-73.329,170.161,32.542,156.139
C06098=1048.763,-33.247,-73.315,170.159,32.541,156.139
C06099=1048.756,-33.496,-73.302,170.157,32.539,156.139
C06100=1048.750,-33.745,-73.289,170.155,32.538,156.139
C06101=1048.744,-33.995,-73.276,170.153,32.536,156.139
C06102=1048.736,-34.343,-73.257,170.150,32.534,156.138
C06103=1048.726,-34.723,-73.237,170.147,32.532,156.138
C06104=1048.719,-35.003,-73.222,170.145,32.530,156.138
C06105=1048.712,-35.283,-73.207,170.143,32.528,156.138
C06106=1048.705,-35.564,-73.192,170.141,32.527,156.137
C06107=1048.698,-35.813,-73.179,170.139,32.525,156.137
C06108=1048.693,-36.063,-73.166,170.137,32.524,156.137
C06109=1048.686,-36.312,-73.153,170.135,32.522,156.137
C06110=1048.680,-36.562,-73.140,170.133,32.521,156.137
C06111=1048.674,-36.812,-73.127,170.131,32.520,156.137
C06112=1048.667,-37.062,-73.114,170.129,32.518,156.136
C06113=1048.662,-37.311,-73.100,170.127,32.517,156.136
C06114=1048.656,-37.560,-73.086,170.126,32.515,156.136
C06115=1048.650,-37.810,-73.074,170.124,32.514,156.136
C06116=1048.644,-38.060,-73.061,170.122,32.513,156.136
C06117=1048.637,-38.309,-73.047,170.120,32.511,156.136
C06118=1048.631,-38.559,-73.034,170.118,32.510,156.135
C06119=1048.625,-38.809,-73.021,170.116,32.508,156.135
C06120=1048.619,-39.059,-73.009,170.114,32.507,156.135
C06121=1048.612,-39.307,-72.996,170.112,32.506,156.135
C06122=1048.606,-39.557,-72.983,170.110,32.504,156.135
C06123=1048.600,-39.807,-72.970,170.108,32.503,156.135
C06124=1048.593,-40.057,-72.956,170.106,32.502,156.134
C06125=1048.587,-40.306,-72.944,170.104,32.500,156.134
C06126=1048.581,-40.556,-72.931,170.102,32.499,156.134
C06127=1048.574,-40.805,-72.918,170.100,32.497,156.134
C06128=1048.568,-41.055,-72.905,170.098,32.496,156.134
C06129=1048.562,-41.304,-72.892,170.096,32.495,156.134
C06130=1048.556,-41.554,-72.880,170.094,32.494,156.133
C06131=1048.549,-41.804,-72.866,170.092,32.492,156.133
C06132=1048.542,-42.053,-72.854,170.090,32.491,156.133
C06133=1048.536,-42.302,-72.841,170.088,32.490,156.133
C06134=1048.530,-42.552,-72.828,170.087,32.488,156.133
C06135=1048.524,-42.802,-72.815,170.085,32.487,156.133
C06136=1048.518,-43.052,-72.802,170.083,32.485,156.133
C06137=1048.511,-43.300,-72.790,170.081,32.484,156.132
C06138=1048.505,-43.550,-72.777,170.079,32.483,156.132
C06139=1048.499,-43.800,-72.764,170.077,32.482,156.132
C06140=1048.492,-44.050,-72.751,170.075,32.480,156.132
C06141=1048.486,-44.299,-72.738,170.073,32.479,156.132
C06142=1048.480,-44.549,-72.726,170.071,32.478,156.132
C06143=1048.474,-44.799,-72.713,170.069,32.476,156.131
C06144=1048.467,-45.048,-72.700,170.066,32.475,156.131
C06145=1048.462,-45.298,-72.687,170.064,32.473,156.131
C06146=1048.455,-45.547,-72.674,170.062,32.473,156.131
C06147=1048.449,-45.797,-72.662,170.060,32.471,156.131
C06148=1048.443,-46.047,-72.650,170.058,32.470,156.131
C06149=1048.437,-46.296,-72.636,170.056,32.468,156.131
C06150=1048.431,-46.546,-72.624,170.054,32.467,156.130
C06151=1048.424,-46.795,-72.611,170.052,32.466,156.130
C06152=1048.418,-47.045,-72.598,170.050,32.464,156.130
C06153=1048.412,-47.295,-72.586,170.049,32.463,156.130
C06154=1048.406,-47.544,-72.573,170.047,32.462,156.130
C06155=1048.400,-47.794,-72.560,170.045,32.461,156.130
C06156=1048.393,-48.043,-72.548,170.043,32.459,156.130
C06157=1048.387,-48.293,-72.535,170.041,32.458,156.129
C06158=1048.381,-48.543,-72.522,170.039,32.457,156.129
C06159=1048.375,-48.792,-72.510,170.037,32.455,156.129
C06160=1048.368,-49.041,-72.497,170.035,32.454,156.129
C06161=1048.362,-49.291,-72.485,170.033,32.453,156.129
C06162=1048.356,-49.541,-72.472,170.031,32.452,156.129
C06163=1048.350,-49.791,-72.459,170.029,32.450,156.129
C06164=1048.343,-50.040,-72.447,170.027,32.449,156.128
C06165=1048.338,-50.290,-72.434,170.025,32.448,156.128
C06166=1048.332,-50.540,-72.422,170.023,32.446,156.128
C06167=1048.324,-50.820,-72.408,170.020,32.445,156.128
C06168=1048.317,-51.102,-72.394,170.018,32.444,156.128
C06169=1048.310,-51.382,-72.380,170.016,32.442,156.128
C06170=1048.303,-51.663,-72.366,170.013,32.441,156.128
C06171=1048.297,-51.913,-72.354,170.011,32.440,156.127
C06172=1048.290,-52.162,-72.342,170.010,32.439,156.127
C06173=1048.284,-52.412,-72.329,170.008,32.438,156.127
C06174=1048.277,-52.662,-72.317,170.006,32.437,156.127
C06175=1048.271,-52.911,-72.305,170.004,32.435,156.127
C06176=1048.265,-53.161,-72.293,170.002,32.435,156.127
C06177=1048.258,-53.411,-72.281,170.000,32.433,156.127
C06178=1048.252,-53.660,-72.267,169.998,32.432,156.127
C06179=1048.245,-53.909,-72.256,169.995,32.431,156.127
C06180=1048.239,-54.159,-72.244,169.993,32.430,156.126
C06181=1048.233,-54.409,-72.231,169.991,32.428,156.126
C06182=1048.226,-54.658,-72.219,169.989,32.428,156.126
C06183=1048.220,-54.908,-72.206,169.987,32.426,156.126
C06184=1048.214,-55.158,-72.195,169.985,32.425,156.126
C06185=1048.207,-55.407,-72.183,169.983,32.424,156.126
C06186=1048.201,-55.657,-72.170,169.981,32.423,156.126
C06187=1048.194,-55.907,-72.158,169.979,32.422,156.126
C06188=1048.189,-56.157,-72.145,169.977,32.421,156.126
C06189=1048.182,-56.406,-72.134,169.975,32.420,156.125
C06190=1048.175,-56.656,-72.122,169.972,32.418,156.125
C06191=1048.169,-56.906,-72.109,169.971,32.417,156.125
C06192=1048.163,-57.155,-72.097,169.969,32.416,156.125
C06193=1048.157,-57.404,-72.085,169.967,32.415,156.125
C06194=1048.151,-57.654,-72.073,169.965,32.414,156.125
C06195=1048.144,-57.904,-72.061,169.963,32.413,156.125
C06196=1048.138,-58.154,-72.048,169.961,32.412,156.125
C06197=1048.132,-58.403,-72.036,169.959,32.411,156.125
C06198=1048.125,-58.653,-72.024,169.957,32.409,156.124
C06199=1048.119,-58.903,-72.012,169.955,32.409,156.124
C06200=1048.113,-59.152,-72.000,169.952,32.407,156.124
C06201=1048.106,-59.401,-71.988,169.950,32.406,156.124
C06202=1048.100,-59.651,-71.976,169.948,32.405,156.124
C06203=1048.094,-59.901,-71.964,169.946,32.404,156.124
C06204=1048.087,-60.151,-71.953,169.944,32.403,156.124
C06205=1048.081,-60.401,-71.940,169.942,32.402,156.124
C06206=1048.075,-60.650,-71.928,169.940,32.401,156.124
C06207=1048.069,-60.899,-71.917,169.938,32.400,156.124
C06208=1048.063,-61.149,-71.904,169.936,32.398,156.123
C06209=1048.056,-61.399,-71.892,169.933,32.397,156.123
C06210=1048.050,-61.648,-71.880,169.932,32.397,156.123
C06211=1048.045,-61.898,-71.869,169.930,32.395,156.123
C06212=1048.038,-62.147,-71.857,169.928,32.394,156.123
C06213=1048.031,-62.397,-71.845,169.926,32.393,156.123
C06214=1048.025,-62.647,-71.832,169.924,32.392,156.123
C06215=1048.019,-62.897,-71.820,169.922,32.391,156.123
C06216=1048.013,-63.145,-71.809,169.920,32.390,156.123
C06217=1048.007,-63.396,-71.797,169.917,32.389,156.123
C06218=1048.000,-63.645,-71.785,169.915,32.388,156.122
C06219=1047.994,-63.895,-71.773,169.913,32.386,156.122
C06220=1047.988,-64.144,-71.761,169.911,32.385,156.122
C06221=1047.982,-64.394,-71.749,169.909,32.385,156.122
C06222=1047.976,-64.644,-71.737,169.907,32.383,156.122
C06223=1047.970,-64.894,-71.725,169.905,32.382,156.122
C06224=1047.964,-65.143,-71.713,169.903,32.381,156.122
C06225=1047.957,-65.393,-71.702,169.901,32.380,156.122
C06226=1047.951,-65.642,-71.690,169.898,32.379,156.122
C06227=1047.945,-65.892,-71.678,169.896,32.378,156.122
C06228=1047.939,-66.142,-71.667,169.894,32.377,156.122
C06229=1047.932,-66.391,-71.655,169.893,32.376,156.121
C06230=1047.926,-66.641,-71.642,169.891,32.375,156.121
C06231=1047.920,-66.923,-71.629,169.888,32.374,156.121
C06232=1047.912,-67.205,-71.616,169.886,32.373,156.121
C06233=1047.906,-67.488,-71.603,169.884,32.372,156.121
C06234=1047.899,-67.770,-71.590,169.881,32.370,156.121
C06235=1047.893,-68.020,-71.577,169.879,32.369,156.121
C06236=1047.886,-68.270,-71.566,169.877,32.368,156.121
C06237=1047.880,-68.519,-71.554,169.875,32.367,156.121
C06238=1047.874,-68.769,-71.543,169.873,32.366,156.121
C06239=1047.868,-69.019,-71.530,169.871,32.365,156.120
C06240=1047.862,-69.268,-71.519,169.868,32.364,156.120
C06241=1047.856,-69.518,-71.508,169.866,32.363,156.120
C06242=1047.850,-69.767,-71.496,169.864,32.362,156.120
C06243=1047.844,-70.017,-71.484,169.862,32.361,156.120
C06244=1047.837,-70.267,-71.472,169.860,32.360,156.120
C06245=1047.831,-70.516,-71.461,169.858,32.359,156.120
C06246=1047.825,-70.766,-71.449,169.856,32.358,156.120
C06247=1047.819,-71.016,-71.437,169.854,32.357,156.120
C06248=1047.813,-71.265,-71.426,169.852,32.356,156.120
C06249=1047.807,-71.515,-71.414,169.850,32.355,156.120
C06250=1047.801,-71.764,-71.403,169.848,32.354,156.119
C06251=1047.795,-72.014,-71.391,169.846,32.353,156.119
C06252=1047.789,-72.264,-71.380,169.844,32.352,156.119
C06253=1047.783,-72.513,-71.368,169.842,32.351,156.119
C06254=1047.776,-72.763,-71.356,169.839,32.350,156.119
C06255=1047.771,-73.013,-71.344,169.837,32.349,156.119
C06256=1047.765,-73.263,-71.333,169.835,32.348,156.119
C06257=1047.759,-73.512,-71.321,169.833,32.347,156.119
C06258=1047.752,-73.762,-71.310,169.831,32.346,156.119
C06259=1047.747,-74.011,-71.299,169.829,32.345,156.119
C06260=1047.740,-74.261,-71.287,169.826,32.344,156.119
C06261=1047.734,-74.511,-71.276,169.824,32.343,156.119
C06262=1047.728,-74.760,-71.265,169.822,32.342,156.119
C06263=1047.721,-75.010,-71.253,169.820,32.341,156.118
C06264=1047.715,-75.260,-71.242,169.818,32.340,156.118
C06265=1047.709,-75.509,-71.230,169.816,32.339,156.118
C06266=1047.703,-75.759,-71.220,169.814,32.339,156.118
C06267=1047.697,-76.009,-71.208,169.812,32.338,156.118
C06268=1047.690,-76.258,-71.196,169.810,32.337,156.118
C06269=1047.684,-76.508,-71.186,169.808,32.336,156.118
C06270=1047.678,-76.758,-71.174,169.806,32.335,156.118
C06271=1047.672,-77.007,-71.163,169.804,32.334,156.118
C06272=1047.666,-77.257,-71.151,169.801,32.333,156.118
C06273=1047.660,-77.507,-71.141,169.799,32.332,156.118
C06274=1047.653,-77.756,-71.129,169.797,32.332,156.118
C06275=1047.648,-78.006,-71.118,169.795,32.331,156.118
C06276=1047.641,-78.256,-71.106,169.793,32.330,156.118
C06277=1047.635,-78.505,-71.096,169.790,32.329,156.118
C06278=1047.629,-78.755,-71.084,169.788,32.328,156.118
C06279=1047.623,-79.005,-71.073,169.786,32.327,156.118
C06280=1047.617,-79.255,-71.062,169.784,32.326,156.117
C06281=1047.611,-79.504,-71.051,169.782,32.325,156.117
C06282=1047.604,-79.754,-71.039,169.779,32.325,156.118
C06283=1047.598,-80.003,-71.028,169.777,32.324,156.117
C06284=1047.592,-80.253,-71.017,169.776,32.323,156.117
C06285=1047.586,-80.503,-71.006,169.774,32.323,156.117
C06286=1047.579,-80.753,-70.995,169.772,32.322,156.117
C06287=1047.573,-81.001,-70.984,169.769,32.321,156.117
C06288=1047.566,-81.252,-70.973,169.767,32.321,156.117
C06289=1047.561,-81.501,-70.962,169.765,32.320,156.117
C06290=1047.554,-81.751,-70.951,169.763,32.319,156.117
C06291=1047.548,-82.000,-70.940,169.761,32.318,156.117
C06292=1047.541,-82.251,-70.929,169.758,32.318,156.117
C06293=1047.536,-82.500,-70.918,169.756,32.317,156.117
C06294=1047.529,-82.750,-70.908,169.754,32.316,156.117
C06295=1047.522,-83.034,-70.895,169.751,32.315,156.117
C06296=1047.515,-83.318,-70.882,169.749,32.314,156.117
C06297=1047.507,-83.603,-70.870,169.746,32.313,156.117
C06298=1047.500,-83.887,-70.857,169.744,32.313,156.117
C06299=1047.494,-84.137,-70.846,169.742,32.312,156.117
C06300=1047.488,-84.387,-70.835,169.739,32.311,156.117
C06301=1047.482,-84.636,-70.825,169.737,32.310,156.117
C06302=1047.475,-84.886,-70.814,169.735,32.310,156.117
C06303=1047.470,-85.136,-70.803,169.734,32.309,156.117
C06304=1047.462,-85.386,-70.792,169.731,32.308,156.117
C06305=1047.457,-85.635,-70.781,169.729,32.308,156.117
C06306=1047.451,-85.885,-70.770,169.727,32.307,156.117
C06307=1047.444,-86.135,-70.760,169.725,32.306,156.117
C06308=1047.438,-86.384,-70.749,169.723,32.305,156.117
C06309=1047.432,-86.634,-70.738,169.720,32.305,156.117
C06310=1047.425,-86.884,-70.727,169.718,32.304,156.117
C06311=1047.420,-87.133,-70.717,169.716,32.303,156.117
C06312=1047.413,-87.383,-70.705,169.714,32.303,156.117
C06313=1047.407,-87.632,-70.695,169.711,32.302,156.117
C06314=1047.401,-87.882,-70.684,169.709,32.301,156.117
C06315=1047.395,-88.132,-70.673,169.707,32.301,156.117
C06316=1047.388,-88.381,-70.663,169.705,32.300,156.116
C06317=1047.382,-88.632,-70.652,169.702,32.299,156.116
C06318=1047.376,-88.882,-70.641,169.700,32.299,156.117
C06319=1047.370,-89.131,-70.631,169.698,32.298,156.116
C06320=1047.364,-89.381,-70.620,169.696,32.297,156.116
C06321=1047.358,-89.630,-70.609,169.694,32.297,156.116
C06322=1047.351,-89.880,-70.598,169.692,32.296,156.116
C06323=1047.345,-90.130,-70.587,169.690,32.295,156.116
C06324=1047.339,-90.379,-70.577,169.688,32.295,156.116
C06325=1047.333,-90.629,-70.567,169.686,32.294,156.116
C06326=1047.327,-90.879,-70.556,169.683,32.294,156.116
C06327=1047.320,-91.128,-70.545,169.681,32.293,156.116
C06328=1047.315,-91.378,-70.534,169.679,32.292,156.116
C06329=1047.309,-91.627,-70.524,169.677,32.292,156.116
C06330=1047.302,-91.877,-70.513,169.674,32.291,156.116
C06331=1047.296,-92.127,-70.503,169.672,32.290,156.116
C06332=1047.291,-92.377,-70.492,169.670,32.290,156.116
C06333=1047.284,-92.626,-70.482,169.668,32.289,156.116
C06334=1047.278,-92.876,-70.470,169.665,32.289,156.116
C06335=1047.272,-93.126,-70.461,169.663,32.288,156.116
C06336=1047.266,-93.376,-70.450,169.661,32.287,156.116
C06337=1047.260,-93.625,-70.439,169.659,32.287,156.116
C06338=1047.253,-93.875,-70.428,169.656,32.286,156.116
C06339=1047.248,-94.125,-70.418,169.654,32.285,156.116
C06340=1047.241,-94.374,-70.408,169.652,32.285,156.116
C06341=1047.235,-94.624,-70.397,169.650,32.284,156.116
C06342=1047.229,-94.875,-70.386,169.648,32.283,156.116
C06343=1047.223,-95.124,-70.376,169.646,32.283,156.116
C06344=1047.217,-95.373,-70.365,169.644,32.282,156.116
C06345=1047.211,-95.622,-70.355,169.642,32.281,156.116
C06346=1047.205,-95.872,-70.345,169.639,32.281,156.116
C06347=1047.199,-96.123,-70.334,169.637,32.280,156.116
C06348=1047.192,-96.372,-70.323,169.635,32.280,156.116
C06349=1047.187,-96.622,-70.313,169.633,32.279,156.116
C06350=1047.181,-96.871,-70.303,169.630,32.279,156.116
C06351=1047.175,-97.121,-70.293,169.628,32.278,156.116
C06352=1047.169,-97.370,-70.282,169.626,32.278,156.116
C06353=1047.162,-97.621,-70.271,169.624,32.277,156.116
C06354=1047.156,-97.870,-70.262,169.621,32.277,156.116
C06355=1047.150,-98.120,-70.251,169.619,32.276,156.116
C06356=1047.144,-98.370,-70.241,169.617,32.275,156.116
C06357=1047.137,-98.620,-70.231,169.615,32.275,156.116
C06358=1047.132,-98.870,-70.220,169.612,32.275,156.116
C06359=1047.125,-99.156,-70.209,169.610,32.274,156.116
C06360=1047.117,-99.442,-70.197,169.607,32.274,156.116
C06361=1047.110,-99.730,-70.186,169.605,32.273,156.116
C06362=1047.103,-100.016,-70.173,169.603,32.272,156.116
C06363=1047.097,-100.265,-70.163,169.601,32.272,156.116
C06364=1047.091,-100.515,-70.154,169.598,32.272,156.116
C06365=1047.084,-100.765,-70.142,169.596,32.271,156.116
C06366=1047.078,-101.015,-70.133,169.594,32.271,156.116
C06367=1047.072,-101.265,-70.123,169.591,32.270,156.117
C06368=1047.066,-101.514,-70.112,169.589,32.270,156.116
C06369=1047.060,-101.764,-70.103,169.587,32.269,156.117
C06370=1047.054,-102.013,-70.093,169.585,32.269,156.117
C06371=1047.048,-102.263,-70.082,169.582,32.268,156.117
C06372=1047.041,-102.513,-70.072,169.580,32.268,156.117
C06373=1047.035,-102.763,-70.062,169.578,32.268,156.117
C06374=1047.029,-103.012,-70.051,169.575,32.267,156.117
C06375=1047.023,-103.262,-70.042,169.573,32.266,156.117
C06376=1047.017,-103.512,-70.032,169.571,32.266,156.117
C06377=1047.010,-103.761,-70.022,169.569,32.266,156.117
C06378=1047.005,-104.011,-70.012,169.566,32.266,156.117
C06379=1046.999,-104.261,-70.002,169.564,32.265,156.117
C06380=1046.992,-104.510,-69.992,169.562,32.265,156.117
C06381=1046.987,-104.760,-69.982,169.560,32.264,156.117
C06382=1046.981,-105.010,-69.972,169.558,32.264,156.117
C06383=1046.974,-105.260,-69.961,169.556,32.264,156.117
C06384=1046.968,-105.510,-69.952,169.554,32.263,156.117
C06385=1046.962,-105.760,-69.942,169.551,32.263,156.117
C06386=1046.956,-106.009,-69.931,169.549,32.262,156.117
C06387=1046.949,-106.259,-69.922,169.547,32.262,156.117
C06388=1046.943,-106.509,-69.912,169.544,32.262,156.117
C06389=1046.938,-106.758,-69.901,169.542,32.262,156.117
C06390=1046.931,-107.008,-69.892,169.540,32.261,156.117
C06391=1046.925,-107.258,-69.882,169.538,32.260,156.117
C06392=1046.919,-107.508,-69.873,169.535,32.260,156.117
C06393=1046.913,-107.757,-69.862,169.533,32.260,156.117
C06394=1046.906,-108.007,-69.853,169.531,32.260,156.117
C06395=1046.901,-108.257,-69.843,169.528,32.259,156.117
C06396=1046.895,-108.507,-69.833,169.526,32.259,156.118
C06397=1046.889,-108.756,-69.824,169.524,32.259,156.118
C06398=1046.882,-109.006,-69.813,169.521,32.259,156.118
C06399=1046.876,-109.255,-69.804,169.519,32.258,156.118
C06400=1046.870,-109.505,-69.794,169.517,32.258,156.118
C06401=1046.864,-109.755,-69.785,169.514,32.258,156.118
C06402=1046.857,-110.005,-69.775,169.513,32.257,156.118
C06403=1046.851,-110.255,-69.765,169.511,32.257,156.118
C06404=1046.846,-110.504,-69.755,169.509,32.257,156.118
C06405=1046.839,-110.754,-69.745,169.506,32.257,156.118
C06406=1046.833,-111.004,-69.735,169.504,32.256,156.118
C06407=1046.827,-111.253,-69.726,169.502,32.256,156.118
C06408=1046.821,-111.503,-69.716,169.499,32.256,156.118
C06409=1046.815,-111.753,-69.707,169.497,32.256,156.118
C06410=1046.809,-112.003,-69.697,169.495,32.255,156.118
C06411=1046.802,-112.253,-69.688,169.492,32.255,156.118
C06412=1046.796,-112.502,-69.678,169.490,32.255,156.118
C06413=1046.790,-112.752,-69.668,169.488,32.255,156.118
C06414=1046.784,-113.001,-69.658,169.485,32.254,156.119
C06415=1046.777,-113.251,-69.649,169.483,32.254,156.119
C06416=1046.771,-113.501,-69.639,169.481,32.254,156.119
C06417=1046.766,-113.751,-69.629,169.479,32.254,156.119
C06418=1046.760,-114.000,-69.620,169.476,32.253,156.119
C06419=1046.754,-114.250,-69.610,169.474,32.253,156.119
C06420=1046.748,-114.500,-69.601,169.472,32.253,156.119
C06421=1046.742,-114.750,-69.591,169.469,32.252,156.119
C06422=1046.735,-114.999,-69.581,169.467,32.252,156.119
C06423=1046.728,-115.286,-69.571,169.465,32.252,156.119
C06424=1046.721,-115.571,-69.561,169.463,32.252,156.119
C06425=1046.714,-115.857,-69.549,169.460,32.252,156.119
C06426=1046.707,-116.142,-69.539,169.457,32.252,156.119
C06427=1046.701,-116.392,-69.529,169.455,32.251,156.119
C06428=1046.695,-116.642,-69.520,169.453,32.251,156.120
C06429=1046.688,-116.892,-69.510,169.450,32.251,156.120
C06430=1046.682,-117.141,-69.501,169.448,32.251,156.120
C06431=1046.677,-117.390,-69.492,169.446,32.251,156.120
C06432=1046.671,-117.640,-69.482,169.443,32.251,156.120
C06433=1046.664,-117.890,-69.472,169.441,32.250,156.120
C06434=1046.658,-118.140,-69.463,169.439,32.250,156.120
C06435=1046.652,-118.390,-69.453,169.436,32.250,156.120
C06436=1046.646,-118.639,-69.444,169.434,32.250,156.120
C06437=1046.640,-118.890,-69.435,169.432,32.250,156.120
C06438=1046.634,-119.139,-69.426,169.429,32.250,156.120
C06439=1046.628,-119.388,-69.417,169.427,32.250,156.120
C06440=1046.621,-119.638,-69.407,169.425,32.250,156.121
C06441=1046.615,-119.888,-69.398,169.422,32.249,156.121
C06442=1046.609,-120.138,-69.388,169.420,32.249,156.121
C06443=1046.603,-120.388,-69.379,169.418,32.250,156.121
C06444=1046.598,-120.637,-69.370,169.415,32.249,156.121
C06445=1046.591,-120.887,-69.360,169.414,32.249,156.121
C06446=1046.585,-121.137,-69.351,169.412,32.249,156.121
C06447=1046.579,-121.387,-69.343,169.409,32.249,156.121
C06448=1046.572,-121.637,-69.333,169.407,32.249,156.121
C06449=1046.567,-121.886,-69.324,169.405,32.249,156.121
C06450=1046.561,-122.136,-69.314,169.402,32.249,156.121
C06451=1046.555,-122.386,-69.305,169.400,32.249,156.122
C06452=1046.548,-122.636,-69.296,169.398,32.248,156.122
C06453=1046.542,-122.885,-69.287,169.395,32.249,156.122
C06454=1046.536,-123.135,-69.278,169.393,32.249,156.122
C06455=1046.530,-123.385,-69.269,169.391,32.248,156.122
C06456=1046.524,-123.635,-69.259,169.388,32.249,156.122
C06457=1046.518,-123.885,-69.250,169.386,32.248,156.122
C06458=1046.512,-124.134,-69.242,169.384,32.248,156.122
C06459=1046.506,-124.384,-69.232,169.381,32.248,156.122
C06460=1046.500,-124.634,-69.223,169.379,32.248,156.122
C06461=1046.494,-124.884,-69.214,169.376,32.248,156.123
C06462=1046.487,-125.133,-69.205,169.374,32.248,156.123
C06463=1046.481,-125.383,-69.196,169.372,32.249,156.123
C06464=1046.475,-125.633,-69.187,169.369,32.248,156.123
C06465=1046.469,-125.882,-69.178,169.367,32.249,156.123
C06466=1046.463,-126.132,-69.169,169.365,32.249,156.123
C06467=1046.457,-126.382,-69.160,169.362,32.249,156.123
C06468=1046.450,-126.631,-69.151,169.361,32.249,156.123
C06469=1046.444,-126.882,-69.142,169.359,32.248,156.123
C06470=1046.439,-127.131,-69.133,169.356,32.249,156.124
C06471=1046.432,-127.381,-69.124,169.354,32.248,156.124
C06472=1046.427,-127.630,-69.115,169.352,32.249,156.124
C06473=1046.420,-127.880,-69.106,169.349,32.248,156.124
C06474=1046.416,-128.129,-69.096,169.347,32.248,156.124
C06475=1046.412,-128.380,-69.086,169.345,32.247,156.124
C06476=1046.408,-128.630,-69.075,169.343,32.246,156.124
C06477=1046.406,-128.880,-69.064,169.341,32.244,156.123
C06478=1046.404,-129.129,-69.051,169.339,32.242,156.123
C06479=1046.404,-129.380,-69.038,169.338,32.239,156.123
C06480=1046.405,-129.630,-69.025,169.336,32.236,156.122
C06481=1046.407,-129.881,-69.011,169.335,32.232,156.122
C06482=1046.409,-130.130,-68.997,169.333,32.228,156.121
C06483=1046.413,-130.381,-68.981,169.333,32.223,156.120
C06484=1046.417,-130.632,-68.966,169.332,32.218,156.119
C06485=1046.423,-130.882,-68.949,169.331,32.212,156.118
C06486=1046.430,-131.132,-68.932,169.330,32.206,156.117
C06487=1046.071,-131.156,-69.170,169.284,32.384,156.150
C06488=1046.065,-130.906,-69.187,169.284,32.389,156.151
C06489=1046.060,-130.656,-69.203,169.285,32.395,156.152
C06490=1046.056,-130.405,-69.219,169.286,32.400,156.153
C06491=1046.052,-130.154,-69.235,169.288,32.405,156.153
C06492=1046.049,-129.905,-69.250,169.289,32.409,156.154
C06493=1046.048,-129.654,-69.263,169.290,32.413,156.155
C06494=1046.047,-129.404,-69.277,169.292,32.416,156.155
C06495=1046.046,-129.154,-69.290,169.294,32.419,156.155
C06496=1046.048,-128.904,-69.302,169.295,32.421,156.156
C06497=1046.050,-128.653,-69.313,169.297,32.423,156.156
C06498=1046.054,-128.403,-69.324,169.298,32.425,156.156
C06499=1046.058,-128.154,-69.335,169.300,32.425,156.156
C06500=1046.063,-127.904,-69.345,169.303,32.426,156.156
C06501=1046.068,-127.654,-69.353,169.305,32.426,156.156
C06502=1046.074,-127.405,-69.363,169.307,32.426,156.156
C06503=1046.081,-127.155,-69.372,169.310,32.426,156.156
C06504=1046.086,-126.905,-69.380,169.312,32.426,156.156
C06505=1046.092,-126.656,-69.390,169.314,32.426,156.156
C06506=1046.098,-126.405,-69.399,169.317,32.426,156.156
C06507=1046.105,-126.156,-69.407,169.319,32.426,156.155
C06508=1046.110,-125.906,-69.416,169.321,32.426,156.155
C06509=1046.117,-125.656,-69.426,169.324,32.426,156.155
C06510=1046.123,-125.407,-69.435,169.326,32.426,156.155
C06511=1046.129,-125.157,-69.443,169.329,32.425,156.155
C06512=1046.135,-124.907,-69.453,169.331,32.426,156.155
C06513=1046.142,-124.658,-69.462,169.333,32.425,156.155
C06514=1046.148,-124.407,-69.470,169.336,32.426,156.155
C06515=1046.153,-124.158,-69.480,169.338,32.425,156.155
C06516=1046.159,-123.908,-69.489,169.340,32.425,156.155
C06517=1046.165,-123.658,-69.498,169.343,32.426,156.154
C06518=1046.172,-123.409,-69.507,169.345,32.425,156.154
C06519=1046.178,-123.159,-69.516,169.347,32.426,156.154
C06520=1046.184,-122.909,-69.525,169.350,32.425,156.154
C06521=1046.190,-122.659,-69.535,169.351,32.425,156.154
C06522=1046.196,-122.409,-69.544,169.353,32.426,156.154
C06523=1046.203,-122.159,-69.552,169.356,32.425,156.154
C06524=1046.208,-121.910,-69.562,169.358,32.426,156.154
C06525=1046.214,-121.660,-69.571,169.361,32.426,156.154
C06526=1046.221,-121.411,-69.581,169.363,32.425,156.153
C06527=1046.226,-121.160,-69.590,169.365,32.426,156.153
C06528=1046.233,-120.910,-69.599,169.368,32.426,156.153
C06529=1046.238,-120.661,-69.608,169.370,32.426,156.153
C06530=1046.245,-120.412,-69.617,169.372,32.426,156.153
C06531=1046.251,-120.162,-69.627,169.375,32.426,156.153
C06532=1046.257,-119.912,-69.636,169.377,32.426,156.153
C06533=1046.263,-119.662,-69.645,169.379,32.426,156.153
C06534=1046.269,-119.413,-69.655,169.382,32.426,156.153
C06535=1046.275,-119.163,-69.664,169.384,32.427,156.153
C06536=1046.281,-118.913,-69.674,169.386,32.426,156.153
C06537=1046.287,-118.663,-69.683,169.389,32.426,156.153
C06538=1046.294,-118.413,-69.692,169.391,32.427,156.152
C06539=1046.300,-118.163,-69.701,169.393,32.427,156.152
C06540=1046.306,-117.914,-69.711,169.396,32.427,156.152
C06541=1046.312,-117.665,-69.720,169.398,32.427,156.152
C06542=1046.318,-117.415,-69.729,169.400,32.427,156.152
C06543=1046.324,-117.165,-69.739,169.403,32.427,156.152
C06544=1046.330,-116.915,-69.749,169.405,32.427,156.152
C06545=1046.337,-116.665,-69.758,169.406,32.427,156.152
C06546=1046.343,-116.416,-69.768,169.409,32.427,156.152
C06547=1046.349,-116.166,-69.777,169.411,32.428,156.152
C06548=1046.356,-115.880,-69.787,169.414,32.428,156.152
C06549=1046.363,-115.594,-69.799,169.416,32.428,156.152
C06550=1046.370,-115.309,-69.809,169.419,32.428,156.151
C06551=1046.377,-115.023,-69.820,169.422,32.428,156.151
C06552=1046.383,-114.773,-69.830,169.424,32.428,156.151
C06553=1046.389,-114.523,-69.839,169.426,32.429,156.151
C06554=1046.395,-114.274,-69.849,169.429,32.429,156.151
C06555=1046.401,-114.024,-69.858,169.431,32.429,156.151
C06556=1046.407,-113.774,-69.868,169.433,32.429,156.151
C06557=1046.413,-113.525,-69.877,169.436,32.429,156.151
C06558=1046.419,-113.275,-69.887,169.438,32.429,156.151
C06559=1046.425,-113.025,-69.896,169.440,32.430,156.151
C06560=1046.432,-112.775,-69.906,169.443,32.430,156.151
C06561=1046.438,-112.525,-69.916,169.445,32.430,156.151
C06562=1046.444,-112.276,-69.925,169.447,32.430,156.151
C06563=1046.450,-112.026,-69.935,169.450,32.431,156.151
C06564=1046.457,-111.777,-69.945,169.452,32.431,156.151
C06565=1046.463,-111.527,-69.955,169.454,32.431,156.150
C06566=1046.469,-111.277,-69.964,169.457,32.431,156.150
C06567=1046.475,-111.027,-69.974,169.458,32.432,156.150
C06568=1046.480,-110.777,-69.984,169.460,32.432,156.150
C06569=1046.487,-110.527,-69.993,169.463,32.432,156.150
C06570=1046.493,-110.277,-70.003,169.465,32.432,156.150
C06571=1046.499,-110.028,-70.013,169.467,32.433,156.150
C06572=1046.505,-109.779,-70.023,169.470,32.433,156.150
C06573=1046.512,-109.529,-70.032,169.472,32.433,156.150
C06574=1046.518,-109.279,-70.042,169.474,32.433,156.150
C06575=1046.524,-109.029,-70.051,169.477,32.434,156.150
C06576=1046.530,-108.779,-70.061,169.479,32.434,156.150
C06577=1046.537,-108.530,-70.071,169.481,32.434,156.150
C06578=1046.542,-108.280,-70.082,169.484,32.435,156.150
C06579=1046.548,-108.030,-70.091,169.486,32.435,156.150
C06580=1046.554,-107.780,-70.101,169.488,32.435,156.150
C06581=1046.561,-107.531,-70.110,169.490,32.435,156.150
C06582=1046.567,-107.281,-70.120,169.493,32.436,156.150
C06583=1046.573,-107.032,-70.130,169.495,32.436,156.149
C06584=1046.579,-106.782,-70.140,169.497,32.436,156.149
C06585=1046.585,-106.532,-70.150,169.500,32.437,156.149
C06586=1046.591,-106.283,-70.160,169.502,32.437,156.149
C06587=1046.597,-106.033,-70.170,169.504,32.437,156.149
C06588=1046.603,-105.783,-70.180,169.507,32.438,156.149
C06589=1046.609,-105.533,-70.190,169.508,32.438,156.149
C06590=1046.616,-105.284,-70.200,169.510,32.438,156.149
C06591=1046.622,-105.034,-70.209,169.513,32.438,156.149
C06592=1046.627,-104.784,-70.220,169.515,32.439,156.149
C06593=1046.634,-104.535,-70.230,169.517,32.440,156.149
C06594=1046.640,-104.284,-70.240,169.519,32.440,156.149
C06595=1046.647,-104.035,-70.250,169.522,32.440,156.149
C06596=1046.652,-103.785,-70.260,169.524,32.440,156.149
C06597=1046.659,-103.535,-70.270,169.526,32.441,156.149
C06598=1046.665,-103.286,-70.280,169.529,32.442,156.149
C06599=1046.670,-103.036,-70.290,169.531,32.442,156.149
C06600=1046.677,-102.787,-70.300,169.533,32.442,156.149
C06601=1046.683,-102.537,-70.310,169.535,32.443,156.149
C06602=1046.689,-102.287,-70.320,169.538,32.443,156.149
C06603=1046.695,-102.037,-70.330,169.540,32.443,156.149
C06604=1046.702,-101.787,-70.340,169.542,32.444,156.149
C06605=1046.707,-101.537,-70.351,169.545,32.445,156.149
C06606=1046.714,-101.288,-70.361,169.547,32.445,156.149
C06607=1046.720,-101.039,-70.371,169.549,32.445,156.149
C06608=1046.726,-100.789,-70.381,169.552,32.445,156.149
C06609=1046.732,-100.539,-70.391,169.554,32.446,156.149
C06610=1046.738,-100.289,-70.401,169.556,32.446,156.149
C06611=1046.745,-100.040,-70.412,169.557,32.447,156.149
C06612=1046.751,-99.753,-70.423,169.560,32.448,156.149
C06613=1046.759,-99.466,-70.435,169.563,32.448,156.149
C06614=1046.766,-99.180,-70.447,169.565,32.448,156.149
C06615=1046.772,-98.892,-70.458,169.568,32.449,156.149
C06616=1046.779,-98.643,-70.469,169.570,32.449,156.149
C06617=1046.785,-98.393,-70.478,169.572,32.449,156.148
C06618=1046.791,-98.143,-70.490,169.575,32.450,156.148
C06619=1046.798,-97.893,-70.499,169.577,32.451,156.148
C06620=1046.804,-97.644,-70.509,169.579,32.451,156.148
C06621=1046.810,-97.395,-70.520,169.582,32.452,156.148
C06622=1046.817,-97.144,-70.530,169.584,32.452,156.148
C06623=1046.822,-96.895,-70.541,169.586,32.452,156.148
C06624=1046.829,-96.645,-70.551,169.588,32.453,156.148
C06625=1046.834,-96.395,-70.562,169.591,32.453,156.148
C06626=1046.840,-96.146,-70.572,169.593,32.454,156.148
C06627=1046.846,-95.896,-70.582,169.595,32.455,156.148
C06628=1046.853,-95.646,-70.593,169.597,32.455,156.148
C06629=1046.859,-95.397,-70.604,169.600,32.456,156.148
C06630=1046.864,-95.147,-70.614,169.602,32.457,156.148
C06631=1046.870,-94.897,-70.625,169.604,32.457,156.148
C06632=1046.877,-94.648,-70.635,169.605,32.458,156.148
C06633=1046.883,-94.397,-70.645,169.608,32.459,156.148
C06634=1046.889,-94.148,-70.656,169.610,32.459,156.148
C06635=1046.895,-93.898,-70.667,169.612,32.460,156.148
C06636=1046.901,-93.649,-70.677,169.614,32.460,156.148
C06637=1046.907,-93.398,-70.687,169.617,32.461,156.148
C06638=1046.913,-93.149,-70.698,169.619,32.461,156.148
C06639=1046.920,-92.900,-70.709,169.621,32.462,156.148
C06640=1046.925,-92.650,-70.719,169.623,32.462,156.148
C06641=1046.931,-92.400,-70.730,169.626,32.463,156.148
C06642=1046.938,-92.150,-70.740,169.628,32.464,156.149
C06643=1046.944,-91.901,-70.751,169.630,32.464,156.148
C06644=1046.950,-91.652,-70.761,169.632,32.465,156.149
C06645=1046.956,-91.401,-70.773,169.635,32.465,156.148
C06646=1046.962,-91.151,-70.783,169.637,32.466,156.149
C06647=1046.968,-90.902,-70.793,169.639,32.466,156.148
C06648=1046.975,-90.652,-70.804,169.641,32.467,156.149
C06649=1046.980,-90.403,-70.815,169.644,32.468,156.149
C06650=1046.987,-90.153,-70.825,169.646,32.468,156.149
C06651=1046.993,-89.903,-70.837,169.648,32.469,156.149
C06652=1046.999,-89.653,-70.847,169.650,32.469,156.149
C06653=1047.005,-89.404,-70.857,169.652,32.470,156.149
C06654=1047.012,-89.154,-70.868,169.654,32.471,156.149
C06655=1047.017,-88.904,-70.879,169.656,32.472,156.149
C06656=1047.024,-88.655,-70.890,169.658,32.472,156.149
C06657=1047.030,-88.405,-70.901,169.661,32.473,156.149
C06658=1047.037,-88.156,-70.911,169.663,32.474,156.149
C06659=1047.042,-87.906,-70.922,169.665,32.474,156.149
C06660=1047.049,-87.656,-70.933,169.667,32.475,156.149
C06661=1047.055,-87.407,-70.943,169.670,32.476,156.149
C06662=1047.061,-87.157,-70.954,169.672,32.476,156.149
C06663=1047.067,-86.907,-70.966,169.674,32.477,156.149
C06664=1047.073,-86.657,-70.975,169.676,32.477,156.149
C06665=1047.080,-86.407,-70.986,169.679,32.478,156.149
C06666=1047.085,-86.158,-70.997,169.681,32.479,156.149
C06667=1047.092,-85.908,-71.008,169.683,32.480,156.149
C06668=1047.098,-85.658,-71.019,169.685,32.480,156.149
C06669=1047.104,-85.409,-71.030,169.687,32.481,156.149
C06670=1047.110,-85.159,-71.041,169.690,32.482,156.149
C06671=1047.117,-84.909,-71.051,169.692,32.482,156.149
C06672=1047.123,-84.660,-71.062,169.694,32.483,156.149
C06673=1047.129,-84.410,-71.074,169.696,32.483,156.149
C06674=1047.136,-84.161,-71.084,169.698,32.484,156.149
C06675=1047.142,-83.911,-71.096,169.700,32.485,156.149
C06676=1047.149,-83.626,-71.108,169.702,32.485,156.149
C06677=1047.156,-83.342,-71.120,169.705,32.486,156.149
C06678=1047.163,-83.057,-71.132,169.707,32.487,156.149
C06679=1047.170,-82.773,-71.145,169.710,32.488,156.149
C06680=1047.176,-82.523,-71.156,169.712,32.489,156.149
C06681=1047.183,-82.274,-71.167,169.714,32.489,156.149
C06682=1047.189,-82.024,-71.178,169.717,32.490,156.149
C06683=1047.195,-81.774,-71.189,169.719,32.491,156.149
C06684=1047.202,-81.525,-71.200,169.721,32.492,156.149
C06685=1047.208,-81.275,-71.211,169.723,32.492,156.149
C06686=1047.214,-81.026,-71.222,169.726,32.493,156.149
C06687=1047.220,-80.775,-71.233,169.728,32.494,156.149
C06688=1047.227,-80.526,-71.244,169.730,32.495,156.149
C06689=1047.233,-80.276,-71.255,169.732,32.495,156.149
C06690=1047.239,-80.026,-71.266,169.734,32.496,156.150
C06691=1047.245,-79.777,-71.277,169.737,32.497,156.150
C06692=1047.253,-79.527,-71.288,169.739,32.498,156.150
C06693=1047.258,-79.278,-71.299,169.741,32.499,156.150
C06694=1047.265,-79.027,-71.310,169.742,32.499,156.150
C06695=1047.271,-78.779,-71.322,169.744,32.500,156.150
C06696=1047.277,-78.528,-71.333,169.747,32.501,156.150
C06697=1047.283,-78.279,-71.344,169.749,32.501,156.150
C06698=1047.289,-78.029,-71.355,169.751,32.502,156.150
C06699=1047.295,-77.780,-71.367,169.753,32.503,156.150
C06700=1047.301,-77.530,-71.378,169.755,32.504,156.150
C06701=1047.307,-77.280,-71.389,169.758,32.505,156.150
C06702=1047.314,-77.031,-71.401,169.760,32.506,156.150
C06703=1047.320,-76.781,-71.412,169.762,32.507,156.150
C06704=1047.326,-76.531,-71.423,169.764,32.507,156.150
C06705=1047.332,-76.282,-71.435,169.766,32.508,156.150
C06706=1047.338,-76.032,-71.446,169.769,32.509,156.150
C06707=1047.344,-75.782,-71.457,169.771,32.510,156.150
C06708=1047.351,-75.533,-71.469,169.773,32.511,156.150
C06709=1047.357,-75.283,-71.480,169.775,32.512,156.151
C06710=1047.363,-75.033,-71.491,169.777,32.513,156.151
C06711=1047.369,-74.784,-71.503,169.779,32.513,156.151
C06712=1047.375,-74.534,-71.514,169.782,32.514,156.151
C06713=1047.381,-74.284,-71.525,169.784,32.515,156.151
C06714=1047.388,-74.034,-71.537,169.786,32.516,156.151
C06715=1047.394,-73.785,-71.548,169.787,32.517,156.151
C06716=1047.401,-73.535,-71.560,169.789,32.518,156.151
C06717=1047.406,-73.286,-71.571,169.792,32.519,156.151
C06718=1047.412,-73.036,-71.583,169.794,32.520,156.151
C06719=1047.418,-72.786,-71.594,169.796,32.521,156.151
C06720=1047.425,-72.537,-71.606,169.798,32.522,156.151
C06721=1047.430,-72.287,-71.617,169.800,32.523,156.151
C06722=1047.437,-72.038,-71.629,169.802,32.524,156.151
C06723=1047.443,-71.787,-71.641,169.804,32.524,156.151
C06724=1047.449,-71.538,-71.652,169.807,32.526,156.152
C06725=1047.455,-71.288,-71.663,169.809,32.527,156.152
C06726=1047.461,-71.039,-71.675,169.811,32.528,156.152
C06727=1047.467,-70.789,-71.687,169.813,32.528,156.152
C06728=1047.473,-70.539,-71.699,169.815,32.529,156.152
C06729=1047.479,-70.290,-71.710,169.817,32.531,156.152
C06730=1047.486,-70.040,-71.722,169.820,32.532,156.152
C06731=1047.491,-69.791,-71.734,169.822,32.533,156.152
C06732=1047.497,-69.541,-71.745,169.824,32.533,156.152
C06733=1047.504,-69.291,-71.757,169.826,32.535,156.152
C06734=1047.510,-69.042,-71.768,169.828,32.536,156.152
C06735=1047.516,-68.792,-71.781,169.830,32.537,156.153
C06736=1047.522,-68.542,-71.792,169.831,32.537,156.153
C06737=1047.528,-68.293,-71.803,169.834,32.538,156.153
C06738=1047.534,-68.043,-71.816,169.836,32.540,156.153
C06739=1047.540,-67.793,-71.827,169.838,32.541,156.153
C06740=1047.547,-67.511,-71.841,169.840,32.542,156.153
C06741=1047.553,-67.229,-71.853,169.843,32.543,156.153
C06742=1047.560,-66.947,-71.867,169.845,32.544,156.153
C06743=1047.568,-66.664,-71.880,169.847,32.545,156.153
C06744=1047.574,-66.414,-71.892,169.850,32.546,156.153
C06745=1047.580,-66.165,-71.904,169.852,32.547,156.153
C06746=1047.587,-65.915,-71.916,169.854,32.548,156.154
C06747=1047.592,-65.665,-71.928,169.856,32.550,156.154
C06748=1047.599,-65.416,-71.940,169.858,32.550,156.154
C06749=1047.605,-65.166,-71.951,169.860,32.551,156.154
C06750=1047.610,-64.916,-71.963,169.862,32.552,156.154
C06751=1047.617,-64.667,-71.975,169.865,32.554,156.154
C06752=1047.624,-64.417,-71.987,169.867,32.554,156.154
C06753=1047.630,-64.168,-71.999,169.869,32.555,156.154
C06754=1047.635,-63.918,-72.010,169.871,32.557,156.154
C06755=1047.642,-63.668,-72.022,169.873,32.558,156.154
C06756=1047.649,-63.419,-72.034,169.874,32.558,156.154
C06757=1047.655,-63.169,-72.047,169.876,32.560,156.155
C06758=1047.661,-62.920,-72.058,169.878,32.561,156.155
C06759=1047.667,-62.670,-72.070,169.881,32.562,156.155
C06760=1047.673,-62.420,-72.082,169.883,32.563,156.155
C06761=1047.679,-62.170,-72.094,169.885,32.564,156.155
C06762=1047.686,-61.921,-72.106,169.887,32.565,156.155
C06763=1047.691,-61.672,-72.118,169.889,32.566,156.155
C06764=1047.698,-61.422,-72.130,169.891,32.567,156.155
C06765=1047.704,-61.172,-72.141,169.893,32.568,156.155
C06766=1047.710,-60.922,-72.154,169.895,32.569,156.155
C06767=1047.717,-60.672,-72.166,169.898,32.570,156.156
C06768=1047.723,-60.424,-72.178,169.900,32.571,156.156
C06769=1047.729,-60.174,-72.190,169.902,32.572,156.156
C06770=1047.736,-59.924,-72.202,169.904,32.574,156.156
C06771=1047.742,-59.675,-72.214,169.906,32.574,156.156
C06772=1047.748,-59.425,-72.227,169.908,32.576,156.156
C06773=1047.754,-59.174,-72.238,169.910,32.577,156.156
C06774=1047.761,-58.926,-72.249,169.912,32.578,156.156
C06775=1047.766,-58.676,-72.262,169.914,32.579,156.156
C06776=1047.773,-58.426,-72.274,169.917,32.580,156.157
C06777=1047.779,-58.176,-72.286,169.919,32.581,156.157
C06778=1047.786,-57.927,-72.298,169.920,32.582,156.157
C06779=1047.792,-57.677,-72.310,169.922,32.583,156.157
C06780=1047.798,-57.427,-72.323,169.924,32.584,156.157
C06781=1047.805,-57.178,-72.335,169.926,32.585,156.157
C06782=1047.811,-56.929,-72.347,169.928,32.586,156.157
C06783=1047.817,-56.679,-72.359,169.930,32.588,156.157
C06784=1047.823,-56.429,-72.371,169.932,32.589,156.157
C06785=1047.829,-56.179,-72.384,169.935,32.589,156.157
C06786=1047.836,-55.930,-72.396,169.937,32.591,156.158
C06787=1047.843,-55.680,-72.408,169.939,32.592,156.158
C06788=1047.849,-55.430,-72.420,169.941,32.593,156.158
C06789=1047.855,-55.181,-72.432,169.943,32.594,156.158
C06790=1047.862,-54.931,-72.444,169.945,32.595,156.158
C06791=1047.868,-54.681,-72.457,169.947,32.596,156.158
C06792=1047.874,-54.432,-72.468,169.949,32.597,156.158
C06793=1047.881,-54.183,-72.482,169.951,32.599,156.158
C06794=1047.887,-53.933,-72.494,169.953,32.600,156.158
C06795=1047.894,-53.683,-72.506,169.955,32.600,156.159
C06796=1047.900,-53.434,-72.518,169.958,32.602,156.159
C06797=1047.906,-53.184,-72.530,169.960,32.603,156.159
C06798=1047.912,-52.934,-72.543,169.962,32.604,156.159
C06799=1047.919,-52.685,-72.555,169.964,32.605,156.159
C06800=1047.925,-52.435,-72.567,169.965,32.607,156.159
C06801=1047.932,-52.185,-72.579,169.967,32.607,156.159
C06802=1047.939,-51.936,-72.592,169.969,32.608,156.159
C06803=1047.944,-51.686,-72.604,169.971,32.610,156.159
C06804=1047.952,-51.406,-72.618,169.974,32.611,156.160
C06805=1047.958,-51.124,-72.631,169.976,32.612,156.160
C06806=1047.966,-50.843,-72.646,169.978,32.614,156.160
C06807=1047.973,-50.563,-72.659,169.981,32.614,156.160
C06808=1047.979,-50.313,-72.672,169.983,32.616,156.160
C06809=1047.985,-50.064,-72.685,169.985,32.617,156.160
C06810=1047.991,-49.814,-72.698,169.987,32.618,156.160
C06811=1047.998,-49.564,-72.709,169.989,32.620,156.161
C06812=1048.004,-49.314,-72.722,169.991,32.621,156.161
C06813=1048.010,-49.065,-72.735,169.993,32.622,156.161
C06814=1048.016,-48.815,-72.748,169.995,32.623,156.161
C06815=1048.023,-48.565,-72.760,169.997,32.625,156.161
C06816=1048.029,-48.316,-72.773,169.999,32.626,156.161
C06817=1048.035,-48.066,-72.786,170.001,32.627,156.161
C06818=1048.041,-47.816,-72.798,170.003,32.629,156.162
C06819=1048.048,-47.567,-72.811,170.005,32.630,156.162
C06820=1048.053,-47.318,-72.823,170.007,32.631,156.162
C06821=1048.059,-47.068,-72.836,170.009,32.632,156.162
C06822=1048.066,-46.818,-72.849,170.010,32.634,156.162
C06823=1048.072,-46.569,-72.861,170.012,32.635,156.162
C06824=1048.078,-46.319,-72.874,170.014,32.636,156.162
C06825=1048.084,-46.070,-72.887,170.016,32.638,156.163
C06826=1048.090,-45.820,-72.900,170.018,32.638,156.163
C06827=1048.096,-45.571,-72.913,170.021,32.640,156.163
C06828=1048.103,-45.321,-72.925,170.023,32.641,156.163
C06829=1048.109,-45.071,-72.937,170.025,32.643,156.163
C06830=1048.115,-44.822,-72.951,170.027,32.644,156.163
C06831=1048.122,-44.571,-72.964,170.029,32.645,156.163
C06832=1048.129,-44.322,-72.976,170.031,32.647,156.164
C06833=1048.135,-44.072,-72.989,170.033,32.648,156.164
C06834=1048.141,-43.823,-73.002,170.035,32.649,156.164
C06835=1048.147,-43.573,-73.015,170.037,32.650,156.164
C06836=1048.153,-43.324,-73.028,170.039,32.652,156.164
C06837=1048.160,-43.074,-73.040,170.041,32.653,156.164
C06838=1048.166,-42.825,-73.053,170.043,32.654,156.164
C06839=1048.172,-42.575,-73.066,170.045,32.656,156.165
C06840=1048.178,-42.326,-73.079,170.047,32.657,156.165
C06841=1048.184,-42.075,-73.092,170.049,32.658,156.165
C06842=1048.191,-41.827,-73.105,170.051,32.659,156.165
C06843=1048.197,-41.577,-73.117,170.053,32.661,156.165
C06844=1048.204,-41.327,-73.130,170.054,32.662,156.165
C06845=1048.209,-41.077,-73.143,170.056,32.663,156.165
C06846=1048.216,-40.828,-73.156,170.058,32.665,156.166
C06847=1048.222,-40.578,-73.169,170.060,32.666,156.166
C06848=1048.229,-40.329,-73.182,170.062,32.668,156.166
C06849=1048.235,-40.079,-73.194,170.064,32.668,156.166
C06850=1048.241,-39.830,-73.208,170.066,32.670,156.166
C06851=1048.247,-39.580,-73.221,170.068,32.671,156.166
C06852=1048.253,-39.330,-73.233,170.070,32.673,156.167
C06853=1048.260,-39.081,-73.247,170.072,32.674,156.167
C06854=1048.267,-38.831,-73.260,170.074,32.675,156.167
C06855=1048.273,-38.582,-73.272,170.076,32.676,156.167
C06856=1048.279,-38.332,-73.286,170.078,32.678,156.167
C06857=1048.285,-38.082,-73.298,170.080,32.679,156.167
C06858=1048.291,-37.833,-73.311,170.082,32.681,156.168
C06859=1048.298,-37.584,-73.325,170.084,32.682,156.168
C06860=1048.303,-37.334,-73.339,170.086,32.684,156.168
C06861=1048.310,-37.084,-73.351,170.088,32.685,156.168
C06862=1048.316,-36.834,-73.365,170.090,32.687,156.168
C06863=1048.322,-36.585,-73.378,170.092,32.687,156.168
C06864=1048.328,-36.335,-73.391,170.094,32.689,156.169
C06865=1048.334,-36.086,-73.404,170.096,32.690,156.169
C06866=1048.341,-35.836,-73.417,170.098,32.692,156.169
C06867=1048.347,-35.587,-73.431,170.100,32.693,156.169
C06868=1048.354,-35.306,-73.445,170.101,32.695,156.169
C06869=1048.361,-35.026,-73.460,170.103,32.697,156.170
C06870=1048.368,-34.745,-73.475,170.106,32.698,156.170
C06871=1048.375,-34.465,-73.490,170.108,32.700,156.170
C06872=1048.381,-34.215,-73.503,170.110,32.701,156.170
C06873=1048.387,-33.966,-73.516,170.112,32.703,156.170
C06874=1048.394,-33.716,-73.530,170.114,32.704,156.170
C06875=1048.400,-33.467,-73.543,170.116,32.706,156.171
C06876=1048.406,-33.217,-73.556,170.118,32.707,156.171
C06877=1048.413,-32.968,-73.569,170.120,32.709,156.171
C06878=1048.418,-32.717,-73.583,170.122,32.710,156.171
C06879=1048.425,-32.468,-73.596,170.124,32.711,156.171
C06880=1048.431,-32.219,-73.609,170.126,32.713,156.172
C06881=1048.437,-31.969,-73.623,170.128,32.714,156.172
C06882=1048.444,-31.719,-73.636,170.130,32.715,156.172
C06883=1048.450,-31.470,-73.650,170.132,32.717,156.172
C06884=1048.456,-31.221,-73.663,170.134,32.718,156.172
C06885=1048.463,-30.971,-73.676,170.136,32.720,156.172
C06886=1048.469,-30.721,-73.689,170.137,32.721,156.173
C06887=1048.475,-30.472,-73.702,170.139,32.722,156.173
C06888=1048.481,-30.222,-73.716,170.141,32.724,156.173
C06889=1048.487,-29.972,-73.730,170.143,32.725,156.173
C06890=1048.494,-29.723,-73.743,170.145,32.727,156.173
C06891=1048.500,-29.474,-73.756,170.147,32.728,156.173
C06892=1048.507,-29.224,-73.770,170.149,32.730,156.174
C06893=1048.513,-28.974,-73.783,170.150,32.731,156.174
C06894=1048.519,-28.725,-73.796,170.152,32.732,156.174
C06895=1048.526,-28.475,-73.810,170.154,32.734,156.174
C06896=1048.531,-28.226,-73.824,170.156,32.735,156.174
C06897=1048.538,-27.976,-73.837,170.158,32.737,156.175
C06898=1048.544,-27.726,-73.851,170.160,32.738,156.175
C06899=1048.551,-27.477,-73.864,170.162,32.740,156.175
C06900=1048.557,-27.227,-73.878,170.164,32.741,156.175
C06901=1048.564,-26.978,-73.891,170.166,32.743,156.175
C06902=1048.569,-26.728,-73.905,170.168,32.744,156.175
C06903=1048.576,-26.478,-73.919,170.170,32.746,156.176
C06904=1048.582,-26.229,-73.932,170.172,32.748,156.176
C06905=1048.588,-25.979,-73.946,170.174,32.749,156.176
C06906=1048.594,-25.730,-73.959,170.175,32.750,156.176
C06907=1048.601,-25.481,-73.973,170.177,32.752,156.176
C06908=1048.606,-25.231,-73.987,170.179,32.753,156.177
C06909=1048.613,-24.981,-74.001,170.181,32.755,156.177
C06910=1048.619,-24.732,-74.015,170.183,32.757,156.177
C06911=1048.625,-24.482,-74.028,170.185,32.758,156.177
C06912=1048.632,-24.233,-74.042,170.187,32.760,156.177
C06913=1048.637,-23.983,-74.055,170.189,32.761,156.178
C06914=1048.643,-23.734,-74.069,170.191,32.763,156.178
C06915=1048.651,-23.484,-74.083,170.193,32.764,156.178
C06916=1048.656,-23.235,-74.097,170.195,32.765,156.178
C06917=1048.663,-22.985,-74.111,170.197,32.768,156.179
C06918=1048.668,-22.735,-74.124,170.198,32.769,156.179
C06919=1048.675,-22.486,-74.138,170.200,32.770,156.179
C06920=1048.682,-22.237,-74.152,170.201,32.772,156.179
C06921=1048.687,-21.987,-74.166,170.203,32.773,156.179
C06922=1048.694,-21.737,-74.180,170.205,32.775,156.179
C06923=1048.700,-21.488,-74.193,170.207,32.777,156.180
C06924=1048.707,-21.238,-74.208,170.209,32.778,156.180
C06925=1048.713,-20.989,-74.221,170.211,32.780,156.180
C06926=1048.718,-20.739,-74.235,170.213,32.781,156.180
C06927=1048.725,-20.489,-74.249,170.215,32.782,156.180
C06928=1048.731,-20.240,-74.263,170.217,32.785,156.181
C06929=1048.738,-19.990,-74.277,170.219,32.786,156.181
C06930=1048.744,-19.741,-74.290,170.220,32.787,156.181
C06931=1048.750,-19.491,-74.304,170.222,32.789,156.181
C06932=1048.757,-19.210,-74.320,170.224,32.791,156.182
C06933=1048.764,-18.929,-74.336,170.227,32.792,156.182
C06934=1048.772,-18.648,-74.351,170.229,32.794,156.182
C06935=1048.779,-18.366,-74.367,170.231,32.796,156.182
C06936=1048.785,-18.116,-74.381,170.233,32.797,156.182
C06937=1048.792,-17.867,-74.395,170.235,32.799,156.183
C06938=1048.797,-17.618,-74.409,170.237,32.801,156.183
C06939=1048.804,-17.368,-74.423,170.238,32.802,156.183
C06940=1048.810,-17.119,-74.437,170.240,32.804,156.183
C06941=1048.817,-16.869,-74.451,170.242,32.805,156.184
C06942=1048.823,-16.619,-74.464,170.244,32.807,156.184
C06943=1048.829,-16.370,-74.479,170.246,32.809,156.184
C06944=1048.835,-16.120,-74.492,170.248,32.810,156.184
C06945=1048.842,-15.871,-74.507,170.250,32.811,156.184
C06946=1048.848,-15.622,-74.521,170.252,32.813,156.185
C06947=1048.854,-15.371,-74.535,170.254,32.814,156.185
C06948=1048.860,-15.150,-74.547,170.254,32.816,156.185
C06949=1048.866,-14.929,-74.560,170.256,32.817,156.185
C06950=1048.870,-14.708,-74.573,170.258,32.819,156.185
C06951=1048.877,-14.486,-74.586,170.259,32.821,156.186
C06952=1048.882,-14.265,-74.597,170.261,32.822,156.186
C06953=1048.887,-14.043,-74.611,170.263,32.823,156.186
C06954=1048.893,-13.822,-74.623,170.264,32.825,156.186
C06955=1048.899,-13.601,-74.636,170.266,32.826,156.186
C06956=1048.904,-13.351,-74.650,170.268,32.828,156.187
C06957=1048.911,-13.102,-74.665,170.270,32.830,156.187
C06958=1048.917,-12.852,-74.678,170.271,32.831,156.187
C06959=1048.923,-12.603,-74.693,170.273,32.832,156.187
C06960=1048.929,-12.353,-74.707,170.275,32.835,156.188
C06961=1048.936,-12.104,-74.721,170.277,32.836,156.188
C06962=1048.942,-11.855,-74.736,170.279,32.837,156.188
C06963=1048.948,-11.604,-74.750,170.281,32.839,156.188
C06964=1048.955,-11.355,-74.764,170.283,32.841,156.188
C06965=1048.960,-11.106,-74.778,170.284,32.842,156.189
C06966=1048.967,-10.856,-74.793,170.286,32.844,156.189
C06967=1048.973,-10.607,-74.806,170.288,32.846,156.189
C06968=1048.979,-10.357,-74.821,170.290,32.847,156.189
C06969=1048.985,-10.108,-74.836,170.292,32.849,156.190
C06970=1048.992,-9.858,-74.849,170.294,32.851,156.190
C06971=1048.998,-9.608,-74.864,170.296,32.852,156.190
C06972=1049.004,-9.359,-74.879,170.297,32.854,156.190
C06973=1049.010,-9.109,-74.893,170.299,32.856,156.190
C06974=1049.017,-8.860,-74.908,170.301,32.858,156.191
C06975=1049.023,-8.611,-74.922,170.303,32.859,156.191
C06976=1049.029,-8.361,-74.936,170.305,32.860,156.191
C06977=1049.036,-8.112,-74.950,170.307,32.863,156.191
C06978=1049.042,-7.862,-74.965,170.309,32.864,156.192
C06979=1049.048,-7.612,-74.980,170.310,32.865,156.192
C06980=1049.054,-7.363,-74.994,170.312,32.867,156.192
C06981=1049.061,-7.114,-75.008,170.313,32.869,156.192
C06982=1049.067,-6.863,-75.023,170.315,32.871,156.193
C06983=1049.073,-6.614,-75.037,170.317,32.872,156.193
C06984=1049.080,-6.365,-75.052,170.319,32.874,156.193
C06985=1049.086,-6.115,-75.067,170.320,32.876,156.193
C06986=1049.092,-5.866,-75.080,170.322,32.877,156.193
C06987=1049.098,-5.616,-75.095,170.324,32.879,156.194
C06988=1049.105,-5.367,-75.110,170.326,32.881,156.194
C06989=1049.111,-5.118,-75.124,170.328,32.882,156.194
C06990=1049.117,-4.868,-75.139,170.330,32.883,156.194
C06991=1049.124,-4.618,-75.153,170.331,32.885,156.195
C06992=1049.131,-4.369,-75.168,170.333,32.887,156.195
C06993=1049.136,-4.120,-75.182,170.335,32.889,156.195
C06994=1049.143,-3.870,-75.197,170.337,32.890,156.195
C06995=1049.149,-3.620,-75.212,170.339,32.892,156.195
C06996=1049.158,-3.282,-75.232,170.341,32.894,156.196
C06997=1049.166,-2.942,-75.252,170.344,32.897,156.196
C06998=1049.174,-2.603,-75.272,170.346,32.899,156.197
C06999=1049.183,-2.264,-75.292,170.349,32.901,156.197
C07000=1049.189,-2.014,-75.307,170.350,32.903,156.197
C07001=1049.195,-1.765,-75.322,170.352,32.905,156.197
C07002=1049.201,-1.515,-75.336,170.354,32.907,156.198
C07003=1049.207,-1.265,-75.351,170.356,32.908,156.198
C07004=1049.213,-1.016,-75.365,170.358,32.910,156.198
C07005=1049.220,-0.766,-75.380,170.359,32.912,156.198
C07006=1049.226,-0.517,-75.395,170.361,32.914,156.199
C07007=1049.232,-0.268,-75.410,170.363,32.916,156.199
C07008=1049.238,-0.018,-75.425,170.365,32.917,156.199
C07009=1049.244,0.231,-75.440,170.367,32.919,156.199
C07010=1049.251,0.481,-75.455,170.368,32.921,156.200
C07011=1049.257,0.730,-75.469,170.370,32.923,156.200
C07012=1049.262,0.980,-75.485,170.372,32.924,156.200
C07013=1049.269,1.230,-75.500,170.374,32.926,156.200
C07014=1049.274,1.479,-75.514,170.376,32.928,156.201
C07015=1049.281,1.728,-75.529,170.377,32.930,156.201
C07016=1049.287,1.978,-75.544,170.378,32.932,156.201
C07017=1049.294,2.228,-75.559,170.380,32.933,156.201
C07018=1049.299,2.477,-75.574,170.382,32.935,156.202
C07019=1049.306,2.726,-75.589,170.383,32.936,156.202
C07020=1049.312,2.975,-75.604,170.385,32.938,156.202
C07021=1049.319,3.225,-75.619,170.387,32.941,156.202
C07022=1049.325,3.475,-75.634,170.389,32.942,156.203
C07023=1049.331,3.724,-75.649,170.391,32.944,156.203
C07024=1049.337,3.973,-75.664,170.392,32.945,156.203
C07025=1049.344,4.223,-75.679,170.394,32.947,156.203
C07026=1049.349,4.473,-75.694,170.396,32.949,156.204
C07027=1049.356,4.723,-75.709,170.398,32.951,156.204
C07028=1049.362,4.971,-75.724,170.400,32.953,156.204
C07029=1049.368,5.221,-75.739,170.401,32.954,156.204
C07030=1049.375,5.470,-75.754,170.403,32.956,156.205
C07031=1049.381,5.720,-75.769,170.405,32.958,156.205
C07032=1049.387,5.969,-75.784,170.407,32.960,156.205
C07033=1049.393,6.218,-75.799,170.408,32.961,156.205
C07034=1049.400,6.468,-75.814,170.410,32.963,156.206
C07035=1049.406,6.718,-75.829,170.412,32.965,156.206
C07036=1049.412,6.967,-75.845,170.414,32.967,156.206
C07037=1049.418,7.217,-75.860,170.416,32.969,156.207
C07038=1049.425,7.466,-75.875,170.417,32.970,156.207
C07039=1049.431,7.716,-75.890,170.419,32.972,156.207
C07040=1049.437,7.965,-75.904,170.421,32.973,156.207
C07041=1049.444,8.214,-75.920,170.423,32.976,156.208
C07042=1049.450,8.464,-75.935,170.424,32.977,156.208
C07043=1049.456,8.713,-75.950,170.426,32.979,156.208
C07044=1049.462,8.963,-75.965,170.428,32.981,156.208
C07045=1049.469,9.212,-75.981,170.430,32.982,156.209
C07046=1049.475,9.462,-75.996,170.431,32.984,156.209
C07047=1049.481,9.712,-76.011,170.433,32.986,156.209
C07048=1049.488,9.961,-76.027,170.435,32.988,156.209
C07049=1049.494,10.210,-76.041,170.437,32.990,156.210
C07050=1049.500,10.459,-76.056,170.439,32.991,156.210
C07051=1049.507,10.709,-76.071,170.440,32.993,156.210
C07052=1049.513,10.958,-76.087,170.442,32.995,156.210
C07053=1049.519,11.208,-76.102,170.444,32.997,156.211
C07054=1049.525,11.458,-76.117,170.446,32.999,156.211
C07055=1049.532,11.707,-76.133,170.447,33.000,156.211
C07056=1049.538,11.956,-76.148,170.449,33.002,156.211
C07057=1049.545,12.206,-76.163,170.451,33.004,156.212
C07058=1049.551,12.455,-76.179,170.453,33.006,156.212
C07059=1049.557,12.705,-76.194,170.454,33.007,156.212
C07060=1049.564,12.990,-76.211,170.456,33.009,156.212
C07061=1049.572,13.275,-76.229,170.458,33.011,156.213
C07062=1049.579,13.559,-76.246,170.459,33.013,156.213
C07063=1049.587,13.844,-76.263,170.461,33.015,156.213
C07064=1049.593,14.093,-76.280,170.463,33.017,156.214
C07065=1049.599,14.343,-76.295,170.465,33.019,156.214
C07066=1049.606,14.593,-76.310,170.467,33.021,156.214
C07067=1049.611,14.842,-76.326,170.468,33.023,156.214
C07068=1049.618,15.092,-76.341,170.470,33.024,156.215
C07069=1049.625,15.341,-76.356,170.472,33.026,156.215
C07070=1049.630,15.591,-76.372,170.474,33.028,156.215
C07071=1049.637,15.840,-76.388,170.475,33.030,156.216
C07072=1049.642,16.089,-76.403,170.477,33.031,156.216
C07073=1049.649,16.338,-76.418,170.479,33.033,156.216
C07074=1049.655,16.588,-76.433,170.481,33.035,156.216
C07075=1049.661,16.837,-76.450,170.482,33.037,156.217
C07076=1049.667,17.087,-76.465,170.484,33.039,156.217
C07077=1049.673,17.336,-76.481,170.486,33.041,156.217
C07078=1049.680,17.585,-76.497,170.487,33.043,156.217
C07079=1049.686,17.835,-76.511,170.489,33.044,156.218
C07080=1049.692,18.084,-76.528,170.491,33.046,156.218
C07081=1049.699,18.334,-76.543,170.493,33.048,156.218
C07082=1049.705,18.583,-76.559,170.494,33.050,156.218
C07083=1049.711,18.833,-76.574,170.496,33.052,156.219
C07084=1049.717,19.082,-76.590,170.498,33.054,156.219
C07085=1049.724,19.331,-76.606,170.500,33.056,156.219
C07086=1049.730,19.581,-76.621,170.501,33.057,156.220
C07087=1049.737,19.831,-76.637,170.503,33.059,156.220
C07088=1049.743,20.081,-76.652,170.505,33.061,156.220
C07089=1049.749,20.330,-76.669,170.506,33.062,156.220
C07090=1049.756,20.579,-76.684,170.508,33.065,156.221
C07091=1049.761,20.829,-76.700,170.510,33.067,156.221
C07092=1049.768,21.078,-76.715,170.512,33.069,156.221
C07093=1049.774,21.327,-76.732,170.513,33.071,156.222
C07094=1049.780,21.577,-76.747,170.515,33.072,156.222
C07095=1049.786,21.826,-76.763,170.517,33.074,156.222
C07096=1049.792,22.076,-76.779,170.518,33.076,156.222
C07097=1049.799,22.325,-76.795,170.520,33.078,156.223
C07098=1049.805,22.575,-76.810,170.522,33.079,156.223
C07099=1049.811,22.824,-76.826,170.524,33.081,156.223
C07100=1049.817,23.073,-76.842,170.525,33.083,156.224
C07101=1049.824,23.323,-76.857,170.527,33.085,156.224
C07102=1049.830,23.572,-76.873,170.529,33.087,156.224
C07103=1049.836,23.821,-76.889,170.530,33.089,156.224
C07104=1049.842,24.070,-76.905,170.532,33.091,156.225
C07105=1049.848,24.320,-76.921,170.534,33.093,156.225
C07106=1049.855,24.570,-76.937,170.536,33.095,156.225
C07107=1049.861,24.820,-76.953,170.537,33.096,156.226
C07108=1049.868,25.069,-76.969,170.539,33.098,156.226
C07109=1049.874,25.318,-76.985,170.541,33.100,156.226
C07110=1049.879,25.568,-77.001,170.542,33.102,156.226
C07111=1049.886,25.817,-77.016,170.544,33.104,156.227
C07112=1049.892,26.066,-77.033,170.546,33.106,156.227
C07113=1049.899,26.315,-77.048,170.548,33.108,156.227
C07114=1049.905,26.565,-77.065,170.549,33.110,156.228
C07115=1049.911,26.815,-77.081,170.551,33.112,156.228
C07116=1049.918,27.064,-77.096,170.553,33.113,156.228
C07117=1049.923,27.314,-77.112,170.554,33.115,156.228
C07118=1049.930,27.563,-77.128,170.556,33.117,156.229
C07119=1049.936,27.812,-77.144,170.558,33.119,156.229
C07120=1049.942,28.061,-77.161,170.559,33.121,156.229
C07121=1049.949,28.311,-77.176,170.561,33.122,156.230
C07122=1049.955,28.561,-77.193,170.563,33.124,156.230
C07123=1049.961,28.810,-77.209,170.565,33.126,156.230
C07124=1049.968,29.095,-77.227,170.566,33.128,156.230
C07125=1049.975,29.382,-77.245,170.568,33.131,156.231
C07126=1049.983,29.669,-77.264,170.570,33.133,156.231
C07127=1049.989,29.954,-77.282,170.572,33.135,156.231
C07128=1049.996,30.204,-77.299,170.574,33.137,156.232
C07129=1050.002,30.453,-77.315,170.576,33.139,156.232
C07130=1050.008,30.703,-77.331,170.577,33.141,156.232
C07131=1050.014,30.952,-77.347,170.579,33.143,156.233
C07132=1050.020,31.201,-77.363,170.581,33.145,156.233
C07133=1050.026,31.451,-77.380,170.582,33.147,156.233
C07134=1050.033,31.701,-77.396,170.584,33.149,156.234
C07135=1050.039,31.950,-77.412,170.586,33.151,156.234
C07136=1050.046,32.199,-77.428,170.587,33.152,156.234
C07137=1050.052,32.448,-77.444,170.589,33.155,156.234
C07138=1050.057,32.698,-77.461,170.590,33.157,156.235
C07139=1050.064,32.946,-77.478,170.592,33.158,156.235
C07140=1050.070,33.196,-77.494,170.593,33.160,156.235
C07141=1050.076,33.446,-77.510,170.595,33.162,156.236
C07142=1050.083,33.695,-77.526,170.596,33.164,156.236
C07143=1050.089,33.944,-77.542,170.598,33.166,156.236
C07144=1050.095,34.194,-77.559,170.600,33.168,156.237
C07145=1050.101,34.444,-77.575,170.601,33.170,156.237
C07146=1050.107,34.693,-77.591,170.603,33.172,156.237
C07147=1050.113,34.942,-77.608,170.605,33.173,156.237
C07148=1050.120,35.191,-77.623,170.607,33.175,156.238
C07149=1050.127,35.441,-77.641,170.608,33.177,156.238
C07150=1050.133,35.690,-77.657,170.610,33.179,156.238
C07151=1050.139,35.939,-77.673,170.612,33.181,156.239
C07152=1050.145,36.189,-77.689,170.613,33.183,156.239
C07153=1050.151,36.439,-77.706,170.615,33.185,156.239
C07154=1050.158,36.688,-77.722,170.617,33.187,156.239
C07155=1050.164,36.937,-77.739,170.618,33.189,156.240
C07156=1050.171,37.187,-77.755,170.620,33.191,156.240
C07157=1050.177,37.436,-77.772,170.622,33.193,156.240
C07158=1050.183,37.685,-77.788,170.623,33.195,156.241
C07159=1050.189,37.935,-77.804,170.625,33.197,156.241
C07160=1050.195,38.184,-77.821,170.627,33.199,156.241
C07161=1050.201,38.434,-77.838,170.628,33.201,156.242
C07162=1050.207,38.683,-77.854,170.630,33.203,156.242
C07163=1050.213,38.932,-77.870,170.632,33.205,156.242
C07164=1050.220,39.182,-77.888,170.633,33.207,156.243
C07165=1050.226,39.431,-77.904,170.635,33.209,156.243
C07166=1050.232,39.680,-77.920,170.637,33.211,156.243
C07167=1050.238,39.929,-77.937,170.638,33.213,156.243
C07168=1050.245,40.179,-77.954,170.640,33.214,156.244
C07169=1050.251,40.428,-77.970,170.642,33.216,156.244
C07170=1050.257,40.677,-77.987,170.643,33.218,156.244
C07171=1050.264,40.927,-78.004,170.645,33.220,156.245
C07172=1050.269,41.177,-78.020,170.647,33.222,156.245
C07173=1050.275,41.426,-78.037,170.648,33.224,156.245
C07174=1050.281,41.675,-78.054,170.650,33.226,156.246
C07175=1050.288,41.925,-78.070,170.651,33.228,156.246
C07176=1050.294,42.174,-78.087,170.653,33.230,156.246
C07177=1050.300,42.423,-78.103,170.655,33.232,156.246
C07178=1050.306,42.673,-78.120,170.656,33.234,156.247
C07179=1050.313,42.922,-78.137,170.658,33.236,156.247
C07180=1050.319,43.171,-78.153,170.660,33.238,156.247
C07181=1050.325,43.421,-78.171,170.661,33.240,156.248
C07182=1050.331,43.670,-78.187,170.663,33.242,156.248
C07183=1050.337,43.920,-78.204,170.665,33.244,156.248
C07184=1050.343,44.169,-78.221,170.666,33.246,156.249
C07185=1050.349,44.418,-78.237,170.668,33.248,156.249
C07186=1050.355,44.667,-78.255,170.670,33.250,156.249
C07187=1050.361,44.918,-78.272,170.671,33.252,156.250
C07188=1050.368,45.203,-78.291,170.673,33.254,156.250
C07189=1050.375,45.489,-78.310,170.675,33.256,156.250
C07190=1050.382,45.775,-78.330,170.677,33.259,156.251
C07191=1050.389,46.062,-78.349,170.679,33.261,156.251
C07192=1050.396,46.311,-78.366,170.680,33.263,156.251
C07193=1050.402,46.560,-78.383,170.682,33.265,156.252
C07194=1050.407,46.809,-78.400,170.684,33.267,156.252
C07195=1050.414,47.059,-78.417,170.685,33.270,156.252
C07196=1050.420,47.308,-78.434,170.687,33.272,156.253
C07197=1050.426,47.557,-78.451,170.689,33.274,156.253
C07198=1050.432,47.807,-78.468,170.690,33.275,156.253
C07199=1050.438,48.056,-78.485,170.692,33.278,156.254
C07200=1050.444,48.306,-78.502,170.693,33.279,156.254
C07201=1050.450,48.555,-78.519,170.695,33.281,156.254
C07202=1050.457,48.804,-78.536,170.697,33.283,156.255
C07203=1050.462,49.053,-78.553,170.698,33.285,156.255
C07204=1050.469,49.303,-78.570,170.700,33.287,156.255
C07205=1050.475,49.552,-78.586,170.702,33.289,156.256
C07206=1050.481,49.802,-78.604,170.703,33.291,156.256
C07207=1050.487,50.051,-78.621,170.705,33.293,156.256
C07208=1050.493,50.300,-78.638,170.707,33.295,156.257
C07209=1050.499,50.550,-78.656,170.708,33.297,156.257
C07210=1050.505,50.798,-78.673,170.710,33.299,156.257
C07211=1050.512,51.049,-78.689,170.711,33.301,156.257
C07212=1050.517,51.298,-78.707,170.713,33.303,156.258
C07213=1050.524,51.547,-78.724,170.715,33.305,156.258
C07214=1050.530,51.796,-78.740,170.716,33.307,156.258
C07215=1050.536,52.045,-78.758,170.718,33.309,156.259
C07216=1050.543,52.295,-78.775,170.720,33.312,156.259
C07217=1050.548,52.544,-78.793,170.721,33.314,156.259
C07218=1050.555,52.794,-78.809,170.723,33.316,156.260
C07219=1050.561,53.043,-78.826,170.725,33.318,156.260
C07220=1050.567,53.292,-78.844,170.726,33.320,156.260
C07221=1050.573,53.541,-78.861,170.728,33.322,156.261
C07222=1050.580,53.791,-78.878,170.730,33.324,156.261
C07223=1050.585,54.040,-78.896,170.732,33.326,156.261
C07224=1050.592,54.290,-78.913,170.734,33.328,156.262
C07225=1050.598,54.539,-78.930,170.735,33.330,156.262
C07226=1050.604,54.789,-78.947,170.737,33.332,156.262
C07227=1050.611,55.037,-78.964,170.739,33.334,156.263
C07228=1050.617,55.287,-78.982,170.740,33.336,156.263
C07229=1050.623,55.536,-78.999,170.742,33.338,156.263
C07230=1050.630,55.785,-79.016,170.744,33.340,156.264
C07231=1050.635,56.035,-79.033,170.745,33.342,156.264
C07232=1050.642,56.284,-79.050,170.747,33.344,156.264
C07233=1050.647,56.533,-79.068,170.749,33.346,156.265
C07234=1050.654,56.783,-79.085,170.750,33.347,156.265
C07235=1050.661,57.032,-79.102,170.752,33.349,156.265
C07236=1050.667,57.281,-79.120,170.753,33.351,156.265
C07237=1050.673,57.531,-79.137,170.755,33.353,156.266
C07238=1050.679,57.780,-79.154,170.757,33.355,156.266
C07239=1050.685,58.029,-79.171,170.758,33.357,156.266
C07240=1050.692,58.279,-79.189,170.760,33.359,156.267
C07241=1050.698,58.528,-79.207,170.762,33.361,156.267
C07242=1050.704,58.777,-79.224,170.763,33.363,156.267
C07243=1050.710,59.027,-79.242,170.765,33.365,156.268
C07244=1050.717,59.276,-79.259,170.767,33.367,156.268
C07245=1050.723,59.525,-79.276,170.768,33.369,156.268
C07246=1050.729,59.774,-79.293,170.770,33.371,156.269
C07247=1050.736,60.023,-79.311,170.771,33.373,156.269
C07248=1050.742,60.274,-79.328,170.773,33.375,156.269
C07249=1050.748,60.523,-79.345,170.775,33.377,156.270
C07250=1050.754,60.772,-79.363,170.776,33.379,156.270
C07251=1050.761,61.022,-79.380,170.778,33.381,156.270
C07252=1050.768,61.307,-79.401,170.780,33.383,156.271
C07253=1050.775,61.593,-79.421,170.782,33.386,156.271
C07254=1050.783,61.879,-79.440,170.784,33.388,156.271
C07255=1050.790,62.165,-79.460,170.786,33.390,156.272
C07256=1050.795,62.414,-79.478,170.787,33.392,156.272
C07257=1050.802,62.663,-79.495,170.789,33.394,156.272
C07258=1050.808,62.913,-79.513,170.791,33.396,156.273
